//Hour pulses
scConnector.scTwilightData.axHours[0]		:= scConnector.scTwilightData.todSystem = TOD#00:00:00 AND scConnector.scTwilightData.dtSystem <> DT#1970-1-1-00:00:00;	//Fix for startup
scConnector.scTwilightData.axHours[1]		:= scConnector.scTwilightData.todSystem = TOD#01:00:00;
scConnector.scTwilightData.axHours[2]		:= scConnector.scTwilightData.todSystem = TOD#02:00:00;
scConnector.scTwilightData.axHours[3]		:= scConnector.scTwilightData.todSystem = TOD#03:00:00;
scConnector.scTwilightData.axHours[4]		:= scConnector.scTwilightData.todSystem = TOD#04:00:00;
scConnector.scTwilightData.axHours[5]		:= scConnector.scTwilightData.todSystem = TOD#05:00:00;
scConnector.scTwilightData.axHours[6]		:= scConnector.scTwilightData.todSystem = TOD#06:00:00;
scConnector.scTwilightData.axHours[7]		:= scConnector.scTwilightData.todSystem = TOD#07:00:00;
scConnector.scTwilightData.axHours[8]		:= scConnector.scTwilightData.todSystem = TOD#08:00:00;
scConnector.scTwilightData.axHours[9]		:= scConnector.scTwilightData.todSystem = TOD#09:00:00;
scConnector.scTwilightData.axHours[10]		:= scConnector.scTwilightData.todSystem = TOD#10:00:00;
scConnector.scTwilightData.axHours[11]		:= scConnector.scTwilightData.todSystem = TOD#11:00:00;
scConnector.scTwilightData.axHours[12]		:= scConnector.scTwilightData.todSystem = TOD#12:00:00;
scConnector.scTwilightData.axHours[13]		:= scConnector.scTwilightData.todSystem = TOD#13:00:00;
scConnector.scTwilightData.axHours[14]		:= scConnector.scTwilightData.todSystem = TOD#14:00:00;
scConnector.scTwilightData.axHours[15]		:= scConnector.scTwilightData.todSystem = TOD#15:00:00;
scConnector.scTwilightData.axHours[16]		:= scConnector.scTwilightData.todSystem = TOD#16:00:00;
scConnector.scTwilightData.axHours[17]		:= scConnector.scTwilightData.todSystem = TOD#17:00:00;
scConnector.scTwilightData.axHours[18]		:= scConnector.scTwilightData.todSystem = TOD#18:00:00;
scConnector.scTwilightData.axHours[19]		:= scConnector.scTwilightData.todSystem = TOD#19:00:00;
scConnector.scTwilightData.axHours[20]		:= scConnector.scTwilightData.todSystem = TOD#20:00:00;
scConnector.scTwilightData.axHours[21]		:= scConnector.scTwilightData.todSystem = TOD#21:00:00;
scConnector.scTwilightData.axHours[22]		:= scConnector.scTwilightData.todSystem = TOD#22:00:00;
scConnector.scTwilightData.axHours[23]		:= scConnector.scTwilightData.todSystem = TOD#23:00:00;
END_ACTION

{attribute 'monitoring' := 'call'} PROPERTY tSlaveErrorResetTime :TIME
SET
tSlaveErrorResetTime_int := tSlaveErrorResetTime;
END_SET
GET
tSlaveErrorResetTime := tSlaveErrorResetTime_int;
END_GET
END_PROPERTY

METHOD Configure_AutoSyncClock
VAR_INPUT
	xAutoSyncClocks		:BOOL := TRUE;		//Sync system time with server
	tAutoSyncClocks		:TIME := T#3H;		//Time for each sync
END_VAR
xAutoSyncClocks_int := xAutoSyncClocks;
tAutoSyncClocks_int := tAutoSyncClocks;
END_METHOD


METHOD Configure_MQTT
VAR_INPUT
	sMQTT_IPAddress				:STRING(15) := '192.168.1.10';
	uiMQTT_ServerPort			:UINT := 1883;
	sMQTT_Username				:STRING(32);
	sMQTT_Password				:STRING(32);
	tMQTT_UpdateTimeOut			:TIME := T#60S;
END_VAR
sMQTT_IPAddress_int := sMQTT_IPAddress;
uiMQTT_ServerPort_int := uiMQTT_ServerPort;
sMQTT_Username_int := sMQTT_Username;
sMQTT_Password_int := sMQTT_Password;
tMQTT_UpdateTimeOut_int := tMQTT_UpdateTimeOut;
END_METHOD

METHOD Configure_HTTP
VAR_INPUT
	sHTTP_IPAddress			:STRING(15) := '192.168.1.10';
	uiHTTP_ServerPort		:UINT := 8080;
END_VAR
sHTTP_IPAddress_int := sHTTP_IPAddress;
uiHTTP_ServerPort_int := uiHTTP_ServerPort;
END_METHOD

METHOD Configure_Twilight
VAR_INPUT
	todSunOffset		:TOD := TOD#00:30:00;	//Time offset (Pre-sunset) / (Post-sunrise)
	todSystemTime_Offset:TOD := TOD#00:00:00;	//Time offset from server to show correct time on system
END_VAR
todSunOffset_int := todSunOffset;
todSystemTime_Offset_int := todSystemTime_Offset;
END_METHOD

{attribute 'monitoring' := 'call'} PROPERTY xAutoReconnect :BOOL
SET
xAutoReconnect_int := xAutoReconnect;
END_SET
GET
xAutoReconnect := xAutoReconnect_int;
END_GET
END_PROPERTY

{attribute 'monitoring' := 'call'} PROPERTY tDataForceSetValues :TIME
SET
tDataForceSetValues_int := tDataForceSetValues;
END_SET
GET
tDataForceSetValues := tDataForceSetValues_int;
END_GET
END_PROPERTY

{attribute 'monitoring' := 'call'} PROPERTY udiUpdateRate_MQTT :UDINT
GET
udiUpdateRate_MQTT := udiUpdateRate_MQTT_int;
END_GET
END_PROPERTY

{attribute 'monitoring' := 'call'} PROPERTY xStartUpDone :BOOL
GET
xStartUpDone := xHTTP_StartUpDone;
END_GET
END_PROPERTY

ACTION ErrorHandling:
//Write error to output
//Sorted on importance	
{warning disable C0327}
//HTTP (1000+)
IF NOT TON_SlaveError_Reset.IN
AND fbHTTP.xError THEN
	scError.xError := TRUE;
	scError.eErrorID := fbHTTP.eErrorID;
	scError.sErrorInstance := _Domoticz_StringExtractAfterDot(sInstanceName);
	sErrorInstance_Concat := '.fbHTTP';
	scError.sErrorInfo := '';
	
//HTTP JSON (3000+)
//Parsing error
ELSIF NOT TON_SlaveError_Reset.IN
AND fbHTTP_Parser.xError THEN
	scError.xError := TRUE;
	scError.eErrorID := fbHTTP_Parser.eErrorID;
	scError.sErrorInstance := _Domoticz_StringExtractAfterDot(sInstanceName);
	sErrorInstance_Concat := '.fbHTTP_Parser';
	scError.sErrorInfo := '';

//HTTP Update timeout
ELSIF NOT TON_SlaveError_Reset.IN
AND TON_HTTP_UpdateTimeOut.Q THEN
	scError.xError := TRUE;
	scError.eErrorID := Domoticz_eErrors.HTTPUpdateTimeOut;
	scError.sErrorInstance := _Domoticz_StringExtractAfterDot(sInstanceName);
	sErrorInstance_Concat := '';
	scError.sErrorInfo := '';
	
//HTTP Connection lost
ELSIF NOT TON_SlaveError_Reset.IN
AND iStepper_HTTP = -10 THEN
	scError.xError := TRUE;
	scError.eErrorID := Domoticz_eErrors.HTTPConnectionLost;
	scError.sErrorInstance := _Domoticz_StringExtractAfterDot(sInstanceName);
	sErrorInstance_Concat := '';
	scError.sErrorInfo := '';
	
//MQTT Receive (2000+)
ELSIF NOT TON_SlaveError_Reset.IN
AND fbMQTT_Receive.xError THEN
	scError.xError := TRUE;
	scError.eErrorID := fbMQTT_Receive.eErrorID;
	scError.sErrorInstance := _Domoticz_StringExtractAfterDot(sInstanceName);
	sErrorInstance_Concat := '.fbMQTT_Receive';
	scError.sErrorInfo := '';
	
//MQTT Send (2000+)
ELSIF NOT TON_SlaveError_Reset.IN
AND fbMQTT_Send.xError THEN
	scError.xError := TRUE;
	scError.eErrorID := fbMQTT_Send.eErrorID;
	scError.sErrorInstance := _Domoticz_StringExtractAfterDot(sInstanceName);
	sErrorInstance_Concat := '.fbMQTT_Send';
	scError.sErrorInfo := '';
	
//MQTT JSON (3000+)
//Error in parsing
ELSIF NOT TON_SlaveError_Reset.IN
AND fbMQTT_Parser.xError THEN
	scError.xError := TRUE;
	scError.eErrorID := fbMQTT_Parser.eErrorID;
	scError.sErrorInstance := _Domoticz_StringExtractAfterDot(sInstanceName);
	sErrorInstance_Concat := '.fbMQTT_Parser';
	scError.sErrorInfo := '';
	
//MQTT Update timeout
ELSIF NOT TON_SlaveError_Reset.IN
AND TON_MQTT_UpdateTimeOut.Q THEN 
	scError.xError := TRUE;
	scError.eErrorID := Domoticz_eErrors.MQTTUpdateTimeOut;
	scError.sErrorInstance := _Domoticz_StringExtractAfterDot(sInstanceName);
	sErrorInstance_Concat := '';
	scError.sErrorInfo := '';
//MQTT Connection lost
ELSIF NOT TON_SlaveError_Reset.IN
AND iStepper_MQTT = -10 THEN 
	scError.xError := TRUE;
	scError.eErrorID := Domoticz_eErrors.MQTTConnectionLost;
	scError.sErrorInstance := _Domoticz_StringExtractAfterDot(sInstanceName);
	sErrorInstance_Concat := '';
	scError.sErrorInfo := '';
{warning restore C0327}

//Error reading data from HTTP object value
ELSIF NOT TON_SlaveError_Reset.IN
AND xHTTP_ObjectError
AND uiHTTP_ObjectError_Source <> 0
AND uiHTTP_ObjectError_wX <> 0 THEN
	scError.xError := TRUE;
	scError.eErrorID := eHTTP_ObjectError;
	scError.sErrorInstance := _Domoticz_StringExtractAfterDot(sInstanceName);
	sErrorInstance_Concat := '';
	sErrorInstance_Concat := CONCAT('.afbHTTP_Object.uiIdentifier[', 	TO_STRING(uiHTTP_ObjectError_Source));
	sErrorInstance_Concat := CONCAT(sErrorInstance_Concat, 				'].uiIdentifier:');
	sErrorInstance_Concat := CONCAT(sErrorInstance_Concat,				TO_STRING(uiHTTP_ObjectError_wX));
	scError.sErrorInfo := '';
	
//Max amount of slaves connected
ELSIF NOT TON_SlaveError_Reset.IN
AND scConnector.uiSlaveTotal = Domoticz_Properties.uiMaxConnectedSlaves THEN
	scError.xError := TRUE;
	scError.eErrorID := Domoticz_eErrors.ObjectMaxReached;
	scError.sErrorInstance := _Domoticz_StringExtractAfterDot(sInstanceName);
	sErrorInstance_Concat := '';
	scError.sErrorInfo := '';
	
//Post server status when booting
ELSIF NOT xHTTP_StartUpDone THEN
	scError.xError := TRUE;
	scError.eErrorID := Domoticz_eErrors.ServerStarting;
	scError.sErrorInstance := _Domoticz_StringExtractAfterDot(sInstanceName);
	sErrorInstance_Concat := '';
	scError.sErrorInfo := '';
	
	//Also write internal state
	scConnector.scSlaveError.xError	:= TRUE;
	scConnector.scSlaveError.eErrorID := Domoticz_eErrors.ServerStarting;
	scConnector.scSlaveError.sErrorInstance := '';
	scConnector.scSlaveError.sErrorInfo := '';
	
//Delete server startup message
ELSIF xHTTP_StartUpDone 
AND scConnector.scSlaveError.xError
AND scConnector.scSlaveError.eErrorID = Domoticz_eErrors.ServerStarting THEN
	scError := scError_Empty;
	scConnector.scSlaveError := scError_Empty;

//(New) error from slave (only when HTTP update is done once and not yet triggered)
ELSIF xHTTP_StartUpDone 
AND scConnector.scSlaveError.xError
AND scConnector.scSlaveError.eErrorID <> Domoticz_eErrors.NoError
AND scConnector.scSlaveError.udiUniqueID = 0
AND NOT TON_SlaveError_Reset.IN THEN
	//Set timer
	TON_SlaveError_Reset.IN := TRUE;
	//Register, check voor empty space
	FOR wX := 1 TO Domoticz_Properties.uiActiveErrors DO
		IF ascActiveSlaveErrors_int[wX].udiUniqueID = 0 THEN
			ascActiveSlaveErrors_int[wX] := scConnector.scSlaveError;
			{warning disable C0371}
			ascActiveSlaveErrors_int[wX].udiUniqueID := TO_UDINT(scConnector.scTwilightData.dtSystem);
			{warning restore C0371}
			scConnector.scSlaveError.udiUniqueID := ascActiveSlaveErrors_int[wX].udiUniqueID;
			EXIT;
		END_IF
	END_FOR
	//End of array reached, no place available
	IF wX = (Domoticz_Properties.uiActiveErrors+1) THEN
		//Return result invalid
		scError.xError := TRUE;
		scError.eErrorID := Domoticz_eErrors.ErrorHandlerArrayFull;
		scError.sErrorInstance := _Domoticz_StringExtractAfterDot(sInstanceName);
		scError.sErrorInfo := '';
		sErrorInstance_Concat := '';
		//scConnector.scSlaveError.udiUniqueID := 0;	//Delete response > no feedback to ErrorInterface FB
	END_IF
	//Output
	scError := scConnector.scSlaveError;	//Copy
	sErrorInstance_Concat := '';	//No additional info
	
//(Remove) error from slave
ELSIF xHTTP_StartUpDone
AND scConnector.scSlaveError.xError
AND scConnector.scSlaveError.eErrorID = Domoticz_eErrors.NoError
AND scConnector.scSlaveError.udiUniqueID <> 0 THEN
	//Unregister, look for ID
	FOR wX := 1 TO Domoticz_Properties.uiActiveErrors DO
		IF ascActiveSlaveErrors_int[wX].udiUniqueID = scConnector.scSlaveError.udiUniqueID THEN
			//Delete entry anyhow
			ascActiveSlaveErrors_int[wX] := scError_Empty;
			//Shift upper array elements
			IF wX <= (Domoticz_Properties.uiActiveErrors-1) THEN
				FOR wY := wX TO (Domoticz_Properties.uiActiveErrors-1) DO
					ascActiveSlaveErrors_int[wY] := ascActiveSlaveErrors_int[wY+1];
				END_FOR
			END_IF
			//Clean last element
			ascActiveSlaveErrors_int[Domoticz_Properties.uiActiveErrors] := scError_Empty;
			EXIT;
		END_IF
	END_FOR
	//End of array reached, not found
	IF wX = (Domoticz_Properties.uiActiveErrors+1) THEN
		//Return result invalid
		scError.xError := TRUE;
		scError.eErrorID := Domoticz_eErrors.ErrorHandlerEntryNotFound;
		scError.sErrorInstance := _Domoticz_StringExtractAfterDot(sInstanceName);
		scError.sErrorInfo := '';
		sErrorInstance_Concat := '';
	END_IF
	//Clear output and connector
	scError := scError_Empty;
	scConnector.scSlaveError := scError_Empty;

//Remove slave error from output after set time
ELSIF xHTTP_StartUpDone 
AND TON_SlaveError_Reset.IN
AND TON_SlaveError_Reset.Q THEN
	//Reset timer
	TON_SlaveError_Reset.IN := FALSE;
	//Clear output and connector
	scError := scError_Empty;
	scConnector.scSlaveError := scError_Empty;
	
//No errors
ELSIF NOT TON_SlaveError_Reset.IN THEN
	scError.xError := FALSE;
	scError.eErrorID := Domoticz_eErrors.NoError;
	scError.sErrorInstance := '';
	sErrorInstance_Concat := '';
	scError.sErrorInfo := '';
END_IF

TON_SlaveError_Reset(IN:=, PT:=tSlaveErrorResetTime_int);	//Run reset timer

//Concat extra source information if available, delete afterwards
psErrorInstance := ADR(scError.sErrorInstance);
psErrorInstance_Concat := ADR(sErrorInstance_Concat);
IF sErrorInstance_Concat <> '' THEN
	StrConcatA(psErrorInstance_Concat, psErrorInstance, SIZEOF(scError.sErrorInstance));
	sErrorInstance_Concat := '';
END_IF
END_ACTION

PROPERTY ascActiveSlaveErrors :ARRAY[1..Domoticz_Properties.uiActiveErrors] OF Domoticz_scError;
GET
ascActiveSlaveErrors := ascActiveSlaveErrors_int;
END_GET
END_PROPERTY

END_FUNCTION_BLOCK

// Function Blocks/Server/_Domoticz_Server_HTTP_Object
{attribute 'conditionalshow_all_locals'}
{attribute 'conditionalshow'}
FUNCTION_BLOCK _Domoticz_Server_HTTP_Object
VAR_INPUT
	sIPAddress					:STRING(15) := '192.168.1.10';
	uiServerPort				:UINT := 8080;
	tTimeOut					:TIME := T#3S;
	dtTimeStamp					:DT;
	xReadData					:BOOL;
	uiIdentifier				:UINT;
END_VAR
VAR_OUTPUT
	xError						:BOOL;
	eErrorID					:Domoticz_eErrors;
	xBusy						:BOOL;
	xDone						:BOOL;
	scObjectData				:Domoticz_scObjectData;
END_VAR
VAR
	//Internal          	
	wX							:WORD;
	xReadData_mem				:BOOL;
	       	
	iStepper					:INT;
	fbHTTP						:SNDLTN_HTTP.HTTP_Client;
	xHTTP_TypeMatched			:BOOL;
	                        	
	xHTTP_DataError				:BOOL;		//Received data contains error
	iHTTP_DataError				:INT;		//Count data errors
	
	//Used for concatting values
	sHTTP_Concat				:STRING(SNDLTN_HTTP.HTTP_Properties.uiHTTPMaxURLSize);
	psHTTP_Concat				:POINTER TO STRING(SNDLTN_HTTP.HTTP_Properties.uiHTTPMaxURLSize);
	sHTTP_ConcatHelper			:STRING(SNDLTN_HTTP.HTTP_Properties.uiHTTPMaxURLSize);
	psHTTP_ConcatHelper			:POINTER TO STRING(SNDLTN_HTTP.HTTP_Properties.uiHTTPMaxURLSize);
	                        	
	//JSON	                	
	fbHTTP_Parser				:SNDLTN_JSON.JSON_Parser;
	fbHTTP_Values				:SNDLTN_JSON.JSON_GetMultiValue;
	
	eHTTP_HumidityStatus		:Domoticz_eHumidityStatus;

END_VAR

Main();

ACTION Main:
{attribute 'conditionalshow'}
CASE iStepper OF

	-10:	//Error
			
		//Reset if needed
		IF NOT xReadData_mem THEN
			xError := FALSE;
			fbHTTP_Parser.xResetError := TRUE;
			iStepper := 0;
		END_IF
	
	0:	//Disabled
		
		//Set outputs if not used
		IF NOT xReadData_mem THEN
			ResetObjectData(); //Empty output
			xBusy := FALSE;
			xDone := FALSE;
		END_IF
		
		//Reset commands
		fbHTTP.xExecute := FALSE;
		fbHTTP_Parser.xResetError := FALSE;
		iHTTP_DataError := 0;
		
		//Wait for command
		IF xReadData AND NOT xReadData_mem
		AND uiIdentifier <> 0 THEN
			xBusy := TRUE;
			iStepper := 10;
		//Invalid identifier
		ELSIF xReadData AND NOT xReadData_mem
		AND uiIdentifier = 0 THEN
			xError := TRUE;
			eErrorID := Domoticz_eErrors.HTTP_InvalidIdentifier;
			iStepper := -10;
		END_IF
		
	10:	//Update object
		
		//Execute and process data
		fbHTTP.xExecute := TRUE;
		DataObject_In();	//Process data
		
		//Wait until processed
		//Not all data received, retrigger
		IF (fbHTTP.xDone AND NOT fbHTTP.xResponseValid) OR xHTTP_DataError THEN
			xHTTP_DataError := FALSE;
			fbHTTP.xExecute := FALSE;
			iHTTP_DataError := iHTTP_DataError + 1;
		//Retrigger max reached, continue (probably invalid ID?)
		ELSIF iHTTP_DataError > 5 THEN
			fbHTTP.xExecute := FALSE;
			xBusy := FALSE;
			xDone := FALSE;
			iStepper := -10;		
		//All data received, continue
		ELSIF fbHTTP.xDone AND fbHTTP.xResponseValid THEN
			fbHTTP.xExecute := FALSE;
			xBusy := FALSE;
			xDone := TRUE;
			iStepper := 0;
		END_IF
		
		//Error occured (outputted in main)
		IF fbHTTP.xError THEN
			xError := TRUE;
			{warning disable C0327}
			eErrorID := fbHTTP.eErrorID;
			{warning restore C0327}
			iStepper := -10;
		ELSIF fbHTTP_Parser.xError THEN
			xError := TRUE;
			eErrorID := Domoticz_eErrors.HTTP_ParsingError;
			iStepper := -10;
		END_IF
	
END_CASE


//HTTP Server
fbHTTP(
	xExecute:= , 
	udiTimeOut:= TIME_TO_UDINT(tTimeOut)*1000, 
);

//Parse HTTP content > only processed if input changes
fbHTTP_Parser(
	xResetError:= , 
	sContent:= fbHTTP.scResponse.sContent, 
);
	
//Get JSON values
fbHTTP_Values(
	pasProperties:= ADR(fbHTTP_Parser.asProperties[0,0]), 
	asPropertyName:= , 
	aeConversionType:= , 
);

//Mem input
xReadData_mem := xReadData;
END_ACTION

METHOD ResetObjectData
VAR_INPUT
END_VAR
scObjectData.uiIdentifier		:= 0;
scObjectData.dtLastUpdate		:= DT#1970-1-1-00:00:00;
scObjectData.dtTimeStamp		:= DT#1970-1-1-00:00:00;
FOR wX := 1 TO Domoticz_Constants.uiMaxSValues DO
	scObjectData.asValue[wX]	:= '';
END_FOR
scObjectData.iValue				:= 0;
scObjectData.eSource			:= _Domoticz_eDataSource.All;
scObjectData.eCommand			:=_Domoticz_eCommandType.Default;
scObjectData.sDeviceType		:= '';
END_METHOD

ACTION DataObject_In:
{attribute 'conditionalshow'}
//HTTP

//Get pointers
psHTTP_Concat := ADR(sHTTP_Concat);
psHTTP_ConcatHelper := ADR(sHTTP_ConcatHelper);

//Construct URL

//HTTP://
sHTTP_Concat := Domoticz_Constants.sURL_HTTP;

//Add server IP
StrConcatA(ADR(sIPAddress), psHTTP_Concat, TO_INT(SNDLTN_HTTP.HTTP_Properties.uiHTTPMaxURLSize));

//Add seperator
sHTTP_ConcatHelper := ':';
StrConcatA(psHTTP_ConcatHelper, psHTTP_Concat, TO_INT(SNDLTN_HTTP.HTTP_Properties.uiHTTPMaxURLSize));

//Add server port
sHTTP_ConcatHelper := TO_STRING(uiServerPort);
StrConcatA(psHTTP_ConcatHelper, psHTTP_Concat, TO_INT(SNDLTN_HTTP.HTTP_Properties.uiHTTPMaxURLSize));

//Add request
StrConcatA(ADR(Domoticz_Constants.sURL_Object), psHTTP_Concat, TO_INT(SNDLTN_HTTP.HTTP_Properties.uiHTTPMaxURLSize));

//Add identifier
sHTTP_ConcatHelper := TO_STRING(uiIdentifier);
StrConcatA(psHTTP_ConcatHelper, psHTTP_Concat, TO_INT(SNDLTN_HTTP.HTTP_Properties.uiHTTPMaxURLSize));

//Get data from HTTP/JSON
fbHTTP.sURL := sHTTP_Concat;
fbHTTP.eRequestType := HTTP_eRequestType.GET;

//Specify data

//Type
fbHTTP_Values.asPropertyName[_Domoticz_eHTTP_PropertyNames.ObjectType] 			:= Domoticz_Constants.sPropertyHTTP_Type;
fbHTTP_Values.aeConversionType[_Domoticz_eHTTP_PropertyNames.ObjectType] 			:= JSON_eConversionType.None;
//Data                                  						                    
fbHTTP_Values.asPropertyName[_Domoticz_eHTTP_PropertyNames.Data] 					:= Domoticz_Constants.sPropertyHTTP_Data;
fbHTTP_Values.aeConversionType[_Domoticz_eHTTP_PropertyNames.Data] 				:= JSON_eConversionType.None;
//SwitchType                            						                    
fbHTTP_Values.asPropertyName[_Domoticz_eHTTP_PropertyNames.SwitchType] 			:= Domoticz_Constants.sPropertyHTTP_SwitchType;
fbHTTP_Values.aeConversionType[_Domoticz_eHTTP_PropertyNames.SwitchType] 			:= JSON_eConversionType.None;
//LastUpdate                            						                    
fbHTTP_Values.asPropertyName[_Domoticz_eHTTP_PropertyNames.LastUpdate] 			:= Domoticz_Constants.sPropertyHTTP_LastUpdate;
fbHTTP_Values.aeConversionType[_Domoticz_eHTTP_PropertyNames.LastUpdate] 			:= JSON_eConversionType.DateAndTime;
                                        						                    
//Level                                 						                    
fbHTTP_Values.asPropertyName[_Domoticz_eHTTP_PropertyNames.Level] 					:= Domoticz_Constants.sPropertyHTTP_Level;
fbHTTP_Values.aeConversionType[_Domoticz_eHTTP_PropertyNames.Level] 				:= JSON_eConversionType.None;
                                        						                                                          						                    
//Additional                            						                    
//Temp+hum+baro                         						                    
//Temperature                           						                    
fbHTTP_Values.asPropertyName[_Domoticz_eHTTP_PropertyNames.Temperature] 			:= Domoticz_Constants.sPropertyHTTP_Temperature;
fbHTTP_Values.aeConversionType[_Domoticz_eHTTP_PropertyNames.Temperature] 			:= JSON_eConversionType.None;
//Humidity                              						                    
fbHTTP_Values.asPropertyName[_Domoticz_eHTTP_PropertyNames.Humidity] 				:= Domoticz_Constants.sPropertyHTTP_Humidity;
fbHTTP_Values.aeConversionType[_Domoticz_eHTTP_PropertyNames.Humidity] 			:= JSON_eConversionType.None;
//Humidity status                           						                    
fbHTTP_Values.asPropertyName[_Domoticz_eHTTP_PropertyNames.HumidityStatus] 		:= Domoticz_Constants.sPropertyHTTP_HumidityStatus;
fbHTTP_Values.aeConversionType[_Domoticz_eHTTP_PropertyNames.HumidityStatus] 		:= JSON_eConversionType.None;
//Barometer                             						                    
fbHTTP_Values.asPropertyName[_Domoticz_eHTTP_PropertyNames.Barometer] 				:= Domoticz_Constants.sPropertyHTTP_Barometer;
fbHTTP_Values.aeConversionType[_Domoticz_eHTTP_PropertyNames.Barometer] 			:= JSON_eConversionType.None;
//Forecast                    						                    
fbHTTP_Values.asPropertyName[_Domoticz_eHTTP_PropertyNames.Forecast] 				:= Domoticz_Constants.sPropertyHTTP_Forecast;
fbHTTP_Values.aeConversionType[_Domoticz_eHTTP_PropertyNames.Forecast] 			:= JSON_eConversionType.None;
//DewPoint                              						                    
fbHTTP_Values.asPropertyName[_Domoticz_eHTTP_PropertyNames.DewPoint] 				:= Domoticz_Constants.sPropertyHTTP_DewPoint;
fbHTTP_Values.aeConversionType[_Domoticz_eHTTP_PropertyNames.DewPoint] 			:= JSON_eConversionType.None;
                                        						                    
//Wind                                  						                    
//Speed                                 						                    
fbHTTP_Values.asPropertyName[_Domoticz_eHTTP_PropertyNames.Speed] 					:= Domoticz_Constants.sPropertyHTTP_Speed;
fbHTTP_Values.aeConversionType[_Domoticz_eHTTP_PropertyNames.Speed] 				:= JSON_eConversionType.None;
//Chill                                 						                    
fbHTTP_Values.asPropertyName[_Domoticz_eHTTP_PropertyNames.Chill] 					:= Domoticz_Constants.sPropertyHTTP_Chill;
fbHTTP_Values.aeConversionType[_Domoticz_eHTTP_PropertyNames.Chill] 				:= JSON_eConversionType.None;
//Gust                                  						                    
fbHTTP_Values.asPropertyName[_Domoticz_eHTTP_PropertyNames.Gust] 					:= Domoticz_Constants.sPropertyHTTP_Gust;
fbHTTP_Values.aeConversionType[_Domoticz_eHTTP_PropertyNames.Gust] 				:= JSON_eConversionType.None;
//Direction                             						                    
fbHTTP_Values.asPropertyName[_Domoticz_eHTTP_PropertyNames.Direction] 				:= Domoticz_Constants.sPropertyHTTP_Direction;
fbHTTP_Values.aeConversionType[_Domoticz_eHTTP_PropertyNames.Direction] 			:= JSON_eConversionType.None;
                                        						                    
//Rain                                  						                    
//Rain                                  						                    
fbHTTP_Values.asPropertyName[_Domoticz_eHTTP_PropertyNames.Rain] 					:= Domoticz_Constants.sPropertyHTTP_Rain;
fbHTTP_Values.aeConversionType[_Domoticz_eHTTP_PropertyNames.Rain] 				:= JSON_eConversionType.None;
//RainRate                              						                    
fbHTTP_Values.asPropertyName[_Domoticz_eHTTP_PropertyNames.RainRate] 				:= Domoticz_Constants.sPropertyHTTP_RainRate;
fbHTTP_Values.aeConversionType[_Domoticz_eHTTP_PropertyNames.RainRate] 			:= JSON_eConversionType.None;
                                        						                    
//RGB(W)(W)                             						                    
//Color                                 						                    
fbHTTP_Values.asPropertyName[_Domoticz_eHTTP_PropertyNames.Color] 					:= Domoticz_Constants.sPropertyHTTP_Color;
fbHTTP_Values.aeConversionType[_Domoticz_eHTTP_PropertyNames.Color] 				:= JSON_eConversionType.None;
                                        						                    
//Energy                                						                    
//Counter cumulative                    						                    
fbHTTP_Values.asPropertyName[_Domoticz_eHTTP_PropertyNames.Counter] 				:= Domoticz_Constants.sPropertyHTTP_Counter;
fbHTTP_Values.aeConversionType[_Domoticz_eHTTP_PropertyNames.Counter] 				:= JSON_eConversionType.None;
//Counter today                     					                        
fbHTTP_Values.asPropertyName[_Domoticz_eHTTP_PropertyNames.CounterToday] 			:= Domoticz_Constants.sPropertyHTTP_CounterToday;
fbHTTP_Values.aeConversionType[_Domoticz_eHTTP_PropertyNames.CounterToday]			:= JSON_eConversionType.None;
//Counter delivery cumulative           						                    
fbHTTP_Values.asPropertyName[_Domoticz_eHTTP_PropertyNames.CounterDelivery] 		:= Domoticz_Constants.sPropertyHTTP_CounterDelivery;
fbHTTP_Values.aeConversionType[_Domoticz_eHTTP_PropertyNames.CounterDelivery] 		:= JSON_eConversionType.None;
//Counter delivery today                  					                        
fbHTTP_Values.asPropertyName[_Domoticz_eHTTP_PropertyNames.CounterDeliveryToday] 	:= Domoticz_Constants.sPropertyHTTP_CounterDeliveryToday;
fbHTTP_Values.aeConversionType[_Domoticz_eHTTP_PropertyNames.CounterDeliveryToday]	:= JSON_eConversionType.None;
//Usage                                 						                    
fbHTTP_Values.asPropertyName[_Domoticz_eHTTP_PropertyNames.Usage] 					:= Domoticz_Constants.sPropertyHTTP_Usage;
fbHTTP_Values.aeConversionType[_Domoticz_eHTTP_PropertyNames.Usage] 				:= JSON_eConversionType.None;
//Usage delivery                        					                        
fbHTTP_Values.asPropertyName[_Domoticz_eHTTP_PropertyNames.UsageDelivery] 			:= Domoticz_Constants.sPropertyHTTP_UsageDelivery;
fbHTTP_Values.aeConversionType[_Domoticz_eHTTP_PropertyNames.UsageDelivery]		:= JSON_eConversionType.None;

//Reset data on start
IF NOT fbHTTP.xDone THEN
	FOR wX := 1 TO Domoticz_Constants.uiMaxSValues DO
		scObjectData.asValue[wX] := '';
	END_FOR		
END_IF
//******************************************************************JSON:PARSE
IF fbHTTP.xDone AND fbHTTP.xResponseValid THEN
		
	scObjectData.uiIdentifier := uiIdentifier;
	
	//Reset data
	FOR wX := 1 TO Domoticz_Constants.uiMaxSValues DO
		scObjectData.asValue[wX] := '';
	END_FOR
	scObjectData.iValue := 0;
	xHTTP_TypeMatched := FALSE;
	
	//Select correct types
	//Switch
	IF fbHTTP_Values.axMatchFound[_Domoticz_eHTTP_PropertyNames.ObjectType] 
	AND (fbHTTP_Values.asPropertyValue[_Domoticz_eHTTP_PropertyNames.ObjectType] = Domoticz_Constants.sType_Lighting1
	OR fbHTTP_Values.asPropertyValue[_Domoticz_eHTTP_PropertyNames.ObjectType] = Domoticz_Constants.sType_Lighting2
	OR fbHTTP_Values.asPropertyValue[_Domoticz_eHTTP_PropertyNames.ObjectType] = Domoticz_Constants.sType_Lighting3
	OR fbHTTP_Values.asPropertyValue[_Domoticz_eHTTP_PropertyNames.ObjectType] = Domoticz_Constants.sType_Lighting4
	OR fbHTTP_Values.asPropertyValue[_Domoticz_eHTTP_PropertyNames.ObjectType] = Domoticz_Constants.sType_Lighting5
	OR fbHTTP_Values.asPropertyValue[_Domoticz_eHTTP_PropertyNames.ObjectType] = Domoticz_Constants.sType_LightSwitch
	OR fbHTTP_Values.asPropertyValue[_Domoticz_eHTTP_PropertyNames.ObjectType] = Domoticz_Constants.sType_Security) THEN
		xHTTP_TypeMatched := TRUE;
		//Selector or selector switch
		IF fbHTTP_Values.axMatchFound[_Domoticz_eHTTP_PropertyNames.SwitchType] 
		AND (fbHTTP_Values.asPropertyValue[_Domoticz_eHTTP_PropertyNames.SwitchType] = Domoticz_Constants.sSwitchType_Selector
		OR fbHTTP_Values.asPropertyValue[_Domoticz_eHTTP_PropertyNames.SwitchType] = Domoticz_Constants.sSwitchType_SelectorSwitch) THEN	
			IF fbHTTP_Values.axMatchFound[_Domoticz_eHTTP_PropertyNames.Level] THEN	//Level
				scObjectData.iValue := 2; 
				scObjectData.asValue[Domoticz_eSValues_General.General] := TO_STRING(_Domoticz_StringToReal(fbHTTP_Values.asPropertyValue[_Domoticz_eHTTP_PropertyNames.Level])); 	//Remove any values				
			ELSIF fbHTTP_Values.axMatchFound[_Domoticz_eHTTP_PropertyNames.Data] THEN	//Data
				scObjectData.iValue := 2; 
				scObjectData.asValue[Domoticz_eSValues_General.General] := TO_STRING(_Domoticz_StringToReal(fbHTTP_Values.asPropertyValue[_Domoticz_eHTTP_PropertyNames.Data])); 	//Remove any values
			END_IF
		//Dimmer
		ELSIF fbHTTP_Values.axMatchFound[_Domoticz_eHTTP_PropertyNames.SwitchType] 
		AND fbHTTP_Values.asPropertyValue[_Domoticz_eHTTP_PropertyNames.SwitchType] = Domoticz_Constants.sSwitchType_Dimmer THEN
			IF fbHTTP_Values.axMatchFound[_Domoticz_eHTTP_PropertyNames.Level] THEN	//Data / Set level
				IF fbHTTP_Values.axMatchFound[_Domoticz_eHTTP_PropertyNames.Data] 
				AND TO_BOOL(_Domoticz_StringToByte(fbHTTP_Values.asPropertyValue[_Domoticz_eHTTP_PropertyNames.Data])) THEN//Dimmer turned off
					scObjectData.iValue := 2; 
					scObjectData.asValue[Domoticz_eSValues_General.General] := TO_STRING(_Domoticz_StringToReal(fbHTTP_Values.asPropertyValue[_Domoticz_eHTTP_PropertyNames.Level])); 	//Remove any values
				ELSE
					IF fbHTTP_Values.axMatchFound[_Domoticz_eHTTP_PropertyNames.Data] THEN		//Data
						scObjectData.iValue := TO_INT(_Domoticz_StringToByte(fbHTTP_Values.asPropertyValue[_Domoticz_eHTTP_PropertyNames.Data])); 
					END_IF
				END_IF
			END_IF
		//None of above
		ELSE	
			IF fbHTTP_Values.axMatchFound[_Domoticz_eHTTP_PropertyNames.Data] THEN 	//Data
				scObjectData.iValue := TO_INT(_Domoticz_StringToByte(fbHTTP_Values.asPropertyValue[_Domoticz_eHTTP_PropertyNames.Data])); 
			END_IF
		END_IF
		
	//RGB(W)(W)
	ELSIF fbHTTP_Values.axMatchFound[_Domoticz_eHTTP_PropertyNames.ObjectType] 
	AND fbHTTP_Values.asPropertyValue[_Domoticz_eHTTP_PropertyNames.ObjectType] = Domoticz_Constants.sType_ColorSwitch THEN
		xHTTP_TypeMatched := TRUE;
		//Color settings
		IF fbHTTP_Values.axMatchFound[_Domoticz_eHTTP_PropertyNames.Color] THEN //Color
			scObjectData.asValue[Domoticz_eSValues_Colors.Red] 			:= _Domoticz_StringExtractColor(fbHTTP_Values.asPropertyValue[_Domoticz_eHTTP_PropertyNames.Color], Domoticz_eSValues_Colors.Red); 
			scObjectData.asValue[Domoticz_eSValues_Colors.Green] 		:= _Domoticz_StringExtractColor(fbHTTP_Values.asPropertyValue[_Domoticz_eHTTP_PropertyNames.Color], Domoticz_eSValues_Colors.Green);
			scObjectData.asValue[Domoticz_eSValues_Colors.Blue] 		:= _Domoticz_StringExtractColor(fbHTTP_Values.asPropertyValue[_Domoticz_eHTTP_PropertyNames.Color], Domoticz_eSValues_Colors.Blue);
			scObjectData.asValue[Domoticz_eSValues_Colors.ColdWhite]	:= _Domoticz_StringExtractColor(fbHTTP_Values.asPropertyValue[_Domoticz_eHTTP_PropertyNames.Color], Domoticz_eSValues_Colors.ColdWhite);
			scObjectData.asValue[Domoticz_eSValues_Colors.WarmWhite]	:= _Domoticz_StringExtractColor(fbHTTP_Values.asPropertyValue[_Domoticz_eHTTP_PropertyNames.Color], Domoticz_eSValues_Colors.WarmWhite);
		END_IF	
		//Brightness level
		IF fbHTTP_Values.axMatchFound[_Domoticz_eHTTP_PropertyNames.Level] THEN //Level (from 0-100 to 0-255)
			scObjectData.asValue[Domoticz_eSValues_Colors.Brightness] := TO_STRING(TRUNC(_Domoticz_StringToReal(fbHTTP_Values.asPropertyValue[_Domoticz_eHTTP_PropertyNames.Level])));
		END_IF
		//Check 'OFF' status
		IF fbHTTP_Values.axMatchFound[_Domoticz_eHTTP_PropertyNames.Data] THEN 
			scObjectData.iValue := TO_INT(TRUNC(_Domoticz_StringToByte(fbHTTP_Values.asPropertyValue[_Domoticz_eHTTP_PropertyNames.Data])));
			IF scObjectData.iValue = 0 THEN	//Force brightness to zero when not enabled
 				scObjectData.asValue[Domoticz_eSValues_Colors.Brightness] := '0.0';
			END_IF
		END_IF
	
	//Temperature / Humidity / Barometer / Dewpoint
	ELSIF fbHTTP_Values.axMatchFound[_Domoticz_eHTTP_PropertyNames.ObjectType] 
	AND (fbHTTP_Values.asPropertyValue[_Domoticz_eHTTP_PropertyNames.ObjectType] = Domoticz_Constants.sType_Temperature
	OR fbHTTP_Values.asPropertyValue[_Domoticz_eHTTP_PropertyNames.ObjectType] = Domoticz_Constants.sType_TemperatureBaro
	OR fbHTTP_Values.asPropertyValue[_Domoticz_eHTTP_PropertyNames.ObjectType] = Domoticz_Constants.sType_TemperatureHumidity
	OR fbHTTP_Values.asPropertyValue[_Domoticz_eHTTP_PropertyNames.ObjectType] = Domoticz_Constants.sType_TemperatureHumidityBaro
	OR fbHTTP_Values.asPropertyValue[_Domoticz_eHTTP_PropertyNames.ObjectType] = Domoticz_Constants.sType_Humidity) THEN
		xHTTP_TypeMatched := TRUE;
		IF fbHTTP_Values.axMatchFound[_Domoticz_eHTTP_PropertyNames.Temperature] THEN	//Temperature
			scObjectData.asValue[Domoticz_eSValues_TempHumBaro.Temperature] := fbHTTP_Values.asPropertyValue[_Domoticz_eHTTP_PropertyNames.Temperature]; 
		END_IF
		IF fbHTTP_Values.axMatchFound[_Domoticz_eHTTP_PropertyNames.Humidity] THEN		//Humidity
			scObjectData.asValue[Domoticz_eSValues_TempHumBaro.Humidity] := fbHTTP_Values.asPropertyValue[_Domoticz_eHTTP_PropertyNames.Humidity]; 
			scObjectData.iValue := TO_INT(_Domoticz_StringToReal(fbHTTP_Values.asPropertyValue[_Domoticz_eHTTP_PropertyNames.Humidity])); 
		END_IF	
		IF fbHTTP_Values.axMatchFound[_Domoticz_eHTTP_PropertyNames.HumidityStatus] THEN	//Humidity Status
			FOR wX := 0 TO 3 DO
				eHTTP_HumidityStatus := TO_INT(wX);
				IF fbHTTP_Values.asPropertyValue[_Domoticz_eHTTP_PropertyNames.HumidityStatus] = TO_STRING(eHTTP_HumidityStatus) THEN
					scObjectData.asValue[Domoticz_eSValues_TempHumBaro.HumidityStatus] := TO_STRING(TO_INT(eHTTP_HumidityStatus));
					EXIT;
				END_IF
			END_FOR
		END_IF
		IF fbHTTP_Values.axMatchFound[_Domoticz_eHTTP_PropertyNames.Barometer] THEN	//Barometer
			scObjectData.asValue[Domoticz_eSValues_TempHumBaro.Barometer] := fbHTTP_Values.asPropertyValue[_Domoticz_eHTTP_PropertyNames.Barometer]; 
		END_IF
		IF fbHTTP_Values.axMatchFound[_Domoticz_eHTTP_PropertyNames.Barometer] THEN	//Forecast
			scObjectData.asValue[Domoticz_eSValues_TempHumBaro.Forecast] := fbHTTP_Values.asPropertyValue[_Domoticz_eHTTP_PropertyNames.Forecast];
		END_IF 
		IF fbHTTP_Values.axMatchFound[_Domoticz_eHTTP_PropertyNames.DewPoint] THEN		//Dewpoint
			scObjectData.asValue[Domoticz_eSValues_TempHumBaro.DewPoint] := fbHTTP_Values.asPropertyValue[_Domoticz_eHTTP_PropertyNames.DewPoint];
		END_IF
		
	//Air Quality
	ELSIF fbHTTP_Values.axMatchFound[_Domoticz_eHTTP_PropertyNames.ObjectType] 
	AND fbHTTP_Values.asPropertyValue[_Domoticz_eHTTP_PropertyNames.ObjectType] = Domoticz_Constants.sType_AirQuality THEN
		xHTTP_TypeMatched := TRUE;
		IF fbHTTP_Values.axMatchFound[_Domoticz_eHTTP_PropertyNames.Data] THEN		//Data
			scObjectData.iValue := TO_INT(_Domoticz_StringToReal(fbHTTP_Values.asPropertyValue[_Domoticz_eHTTP_PropertyNames.Data])); 
		END_IF
		
	//Wind	
	ELSIF fbHTTP_Values.axMatchFound[_Domoticz_eHTTP_PropertyNames.ObjectType] 
	AND fbHTTP_Values.asPropertyValue[_Domoticz_eHTTP_PropertyNames.ObjectType] = Domoticz_Constants.sType_Wind THEN
		xHTTP_TypeMatched := TRUE;
		IF fbHTTP_Values.axMatchFound[_Domoticz_eHTTP_PropertyNames.Speed] THEN 	//Speed
			scObjectData.asValue[Domoticz_eSValues_Wind.Speed] := fbHTTP_Values.asPropertyValue[_Domoticz_eHTTP_PropertyNames.Speed]; 
		END_IF
		IF fbHTTP_Values.axMatchFound[_Domoticz_eHTTP_PropertyNames.Chill] THEN	//Chill
			scObjectData.asValue[Domoticz_eSValues_Wind.Chill] := fbHTTP_Values.asPropertyValue[_Domoticz_eHTTP_PropertyNames.Chill]; 
		END_IF
		IF fbHTTP_Values.axMatchFound[_Domoticz_eHTTP_PropertyNames.Gust] THEN 	//Gust
			scObjectData.asValue[Domoticz_eSValues_Wind.Gust] := fbHTTP_Values.asPropertyValue[_Domoticz_eHTTP_PropertyNames.Gust]; 
		END_IF
		IF fbHTTP_Values.axMatchFound[_Domoticz_eHTTP_PropertyNames.Direction] THEN	//Direction
			scObjectData.asValue[5] := fbHTTP_Values.asPropertyValue[_Domoticz_eHTTP_PropertyNames.Direction]; 
		END_IF	
		
	//Rain
	ELSIF fbHTTP_Values.axMatchFound[_Domoticz_eHTTP_PropertyNames.ObjectType] 
	AND fbHTTP_Values.asPropertyValue[_Domoticz_eHTTP_PropertyNames.ObjectType] = Domoticz_Constants.sType_Rain THEN
		xHTTP_TypeMatched := TRUE;
		IF fbHTTP_Values.axMatchFound[_Domoticz_eHTTP_PropertyNames.Rain] THEN 	//Rain
			scObjectData.asValue[Domoticz_eSValues_Rain.Rain] := fbHTTP_Values.asPropertyValue[_Domoticz_eHTTP_PropertyNames.Rain]; 
		END_IF
		IF fbHTTP_Values.axMatchFound[_Domoticz_eHTTP_PropertyNames.RainRate] THEN 	//Rain rate
			scObjectData.asValue[Domoticz_eSValues_Rain.RainRate] := fbHTTP_Values.asPropertyValue[_Domoticz_eHTTP_PropertyNames.RainRate]; 
		END_IF	
		
	//P1 Smart Meter
	ELSIF (fbHTTP_Values.axMatchFound[_Domoticz_eHTTP_PropertyNames.ObjectType] 
	AND fbHTTP_Values.asPropertyValue[_Domoticz_eHTTP_PropertyNames.ObjectType] = Domoticz_Constants.sType_P1SmartMeter) THEN
		xHTTP_TypeMatched := TRUE;
		IF fbHTTP_Values.axMatchFound[_Domoticz_eHTTP_PropertyNames.Counter] THEN 	//Power cumulative
			scObjectData.asValue[Domoticz_eSValues_P1.Usage1Cumulative] := fbHTTP_Values.asPropertyValue[_Domoticz_eHTTP_PropertyNames.Counter]; 
		END_IF
		IF fbHTTP_Values.axMatchFound[_Domoticz_eHTTP_PropertyNames.CounterToday] THEN 	//Power today
			scObjectData.asValue[Domoticz_eSValues_P1.UsageToday] := fbHTTP_Values.asPropertyValue[_Domoticz_eHTTP_PropertyNames.CounterToday]; 
		END_IF
		IF fbHTTP_Values.axMatchFound[_Domoticz_eHTTP_PropertyNames.CounterDelivery] THEN 	//Power delivery cumulative
			scObjectData.asValue[Domoticz_eSValues_P1.Return1Cumulative] := fbHTTP_Values.asPropertyValue[_Domoticz_eHTTP_PropertyNames.CounterDelivery]; 
		END_IF
		IF fbHTTP_Values.axMatchFound[_Domoticz_eHTTP_PropertyNames.CounterDeliveryToday] THEN 	//Power delivery today
			scObjectData.asValue[Domoticz_eSValues_P1.ReturnToday] := fbHTTP_Values.asPropertyValue[_Domoticz_eHTTP_PropertyNames.CounterDeliveryToday];
		END_IF 
		IF fbHTTP_Values.axMatchFound[_Domoticz_eHTTP_PropertyNames.Usage] THEN 	//Usage
			scObjectData.asValue[Domoticz_eSValues_P1.UsageActual] := fbHTTP_Values.asPropertyValue[_Domoticz_eHTTP_PropertyNames.Usage]; 
		END_IF
		IF fbHTTP_Values.axMatchFound[_Domoticz_eHTTP_PropertyNames.UsageDelivery] THEN 	//Usage delivery
			scObjectData.asValue[Domoticz_eSValues_P1.ReturnActual] := fbHTTP_Values.asPropertyValue[_Domoticz_eHTTP_PropertyNames.UsageDelivery]; 
		END_IF
		
	//General / other
	ELSIF fbHTTP_Values.axMatchFound[_Domoticz_eHTTP_PropertyNames.ObjectType] 
	AND fbHTTP_Values.asPropertyValue[_Domoticz_eHTTP_PropertyNames.ObjectType] = Domoticz_Constants.sType_General THEN
		
		//SubType is available, but not used
		//If usage type found, subtype is presumably kWh or Gas > Electric (counter+instant)
		//Differs from P1, because otherwise MQTT messages are also off (they come in only at 1 and 2)
		IF fbHTTP_Values.axMatchFound[_Domoticz_eHTTP_PropertyNames.Usage] THEN
			xHTTP_TypeMatched := TRUE;
			IF fbHTTP_Values.axMatchFound[_Domoticz_eHTTP_PropertyNames.Usage] THEN 	//Usage
				scObjectData.asValue[Domoticz_eSValues_Usage.Usage] := fbHTTP_Values.asPropertyValue[_Domoticz_eHTTP_PropertyNames.Usage]; 
			END_IF
			IF fbHTTP_Values.axMatchFound[_Domoticz_eHTTP_PropertyNames.Counter] THEN 	//Counter
				scObjectData.asValue[Domoticz_eSValues_Usage.UsageCumulative] := fbHTTP_Values.asPropertyValue[_Domoticz_eHTTP_PropertyNames.Counter]; 
			ELSIF fbHTTP_Values.axMatchFound[_Domoticz_eHTTP_PropertyNames.Data] THEN 	//Counter
				scObjectData.asValue[Domoticz_eSValues_Usage.UsageCumulative] := fbHTTP_Values.asPropertyValue[_Domoticz_eHTTP_PropertyNames.Data]; 
			END_IF
			IF fbHTTP_Values.axMatchFound[_Domoticz_eHTTP_PropertyNames.CounterToday] THEN //Usage today
				scObjectData.asValue[Domoticz_eSValues_Usage.UsageToday] := fbHTTP_Values.asPropertyValue[_Domoticz_eHTTP_PropertyNames.CounterToday]; 
			END_IF
		//Other general types
		ELSE
			xHTTP_TypeMatched := FALSE;
			IF fbHTTP_Values.axMatchFound[_Domoticz_eHTTP_PropertyNames.Data] THEN 
				scObjectData.asValue[Domoticz_eSValues_General.General] := fbHTTP_Values.asPropertyValue[_Domoticz_eHTTP_PropertyNames.Data];
			END_IF	//Data
		END_IF
		
	//Other type > just pass data
	ELSIF fbHTTP_Values.axMatchFound[_Domoticz_eHTTP_PropertyNames.ObjectType] THEN
		xHTTP_TypeMatched := FALSE;
		IF fbHTTP_Values.axMatchFound[_Domoticz_eHTTP_PropertyNames.Data] THEN 
			scObjectData.asValue[Domoticz_eSValues_General.General] := fbHTTP_Values.asPropertyValue[_Domoticz_eHTTP_PropertyNames.Data]; 
		END_IF	//Data
				
	//No type available
	ELSIF NOT fbHTTP_Values.axMatchFound[_Domoticz_eHTTP_PropertyNames.ObjectType] THEN
		xHTTP_DataError := TRUE;
	END_IF

	//Add last update
	IF fbHTTP_Values.axMatchFound[_Domoticz_eHTTP_PropertyNames.LastUpdate] THEN
		scObjectData.dtLastUpdate := fbHTTP_Values.adtPropertyValue[_Domoticz_eHTTP_PropertyNames.LastUpdate];
	ELSE
		scObjectData.dtLastUpdate := DT#1970-1-1-0:0:0;
	END_IF
	
	//Convert data so it has max. two decimals at the end
	IF xHTTP_TypeMatched THEN
		FOR wX := 1 TO Domoticz_Constants.uiMaxSValues DO
			IF scObjectData.asValue[wX] <> '' THEN
				scObjectData.asValue[wX] := TO_STRING(_Domoticz_RoundDecimals(TO_REAL(scObjectData.asValue[wX]),2));
			END_IF
		END_FOR		
	END_IF
			
	//Add info
	scObjectData.sDeviceType := fbHTTP_Values.asPropertyValue[_Domoticz_eHTTP_PropertyNames.ObjectType];	//Transfer type
	scObjectData.dtTimeStamp := dtTimeStamp;	//Add timestamp
	scObjectData.eSource := _Domoticz_eDataSource.HTTP;	//Source is HTTP
	
END_IF
END_ACTION

END_FUNCTION_BLOCK

// Functions/_Domoticz_StringExtractColor
{attribute 'conditionalshow_all_locals'}
{attribute 'conditionalshow'}
FUNCTION _Domoticz_StringExtractColor :STRING(Domoticz_Constants.uiMaxSValuesize)
VAR_INPUT
	sData		:STRING(Domoticz_Constants.uiMaxSValuesize);
	eColor		:Domoticz_eSValues_Colors;
END_VAR
VAR
	//Data processing
	psData		:POINTER TO STRING(Domoticz_Constants.uiMaxSValuesize);
	sSearch		:STRING(2);
	psSearch	:POINTER TO STRING(2);
	sExtract	:STRING(3);
	psExtract	:POINTER TO STRING(4);		//255 + Closing
	
	//Positions
	iPosColor	:INT;
	iPosColom	:INT;
	iPosComma	:INT;
	iPosAccolade:INT;
END_VAR

//Format:
//{\"b\":84,\"cw\":0,\"g\":188,\"m\":3,\"r\":254,\"t\":0,\"ww\":0}

IF eColor >= Domoticz_eSValues_Colors.Red AND eColor <= TO_INT(Domoticz_eSValues_Colors.WarmWhite)
AND sData <> '' THEN

	psData := ADR(sData);
	psSearch := ADR(sSearch);
	psExtract := ADR(sExtract);
	
	//Find position of text
	sSearch := Domoticz_Constants.asProperty_Colors[eColor];
	iPosColor := StrFindA(psData, psSearch, TO_UINT(0));	//Find pos of text
	
	//Find position of colom
	sSearch := ':';
	iPosColom := StrFindA(psData, psSearch, TO_UINT(iPosColor));	//Find pos of colom
	
	//Find position of comma
	sSearch := ',';
	iPosComma := StrFindA(psData, psSearch, TO_UINT(iPosColom));	//Find pos of comma
	
	//Find position of accolade
	sSearch := '}';
	iPosAccolade := StrFindA(psData, psSearch, TO_UINT(iPosColom));	//Find pos of accolade
	
	//Extract data
	//Comma present
	IF iPosComma > 0 THEN
		StrMidA(psData, Domoticz_Constants.uiMaxSValuesize, (iPosComma-iPosColom-1), iPosColom+1,  psExtract, 4);
	//Accolade present
	ELSIF iPosAccolade > 0 THEN
		StrMidA(psData, Domoticz_Constants.uiMaxSValuesize, (iPosAccolade-iPosColom-1), iPosColom+1,  psExtract, 4);
	//Extract last bit
	ELSE
		StrMidA(psData, Domoticz_Constants.uiMaxSValuesize, TO_INT(StrLenA(psData)-iPosColom-1), iPosColom+1,  psExtract, 4);
	END_IF
	StrTrimA(psExtract);
	
	//Output
	_Domoticz_StringExtractColor := sExtract;
	
ELSE
	_Domoticz_StringExtractColor := '';
END_IF

END_FUNCTION

// Functions/_Domoticz_StringExtractAfterDot
{attribute 'conditionalshow_all_locals'}
{attribute 'conditionalshow'}
FUNCTION _Domoticz_StringExtractAfterDot :STRING(Domoticz_Constants.uiInstanceName);
VAR_INPUT
	sData		:STRING(Domoticz_Constants.uiInstanceName);
END_VAR
VAR
	psData		:POINTER TO STRING(Domoticz_Constants.uiInstanceName);
	sFind		:STRING(Domoticz_Constants.uiInstanceName);	
	psFind		:POINTER TO STRING(Domoticz_Constants.uiInstanceName);
	sExtract	:STRING(Domoticz_Constants.uiInstanceName);	
	psExtract	:POINTER TO STRING(Domoticz_Constants.uiInstanceName);	
	
	byDotLoop	:BYTE;
	uiFindDot	:UINT;
	uiLastDot	:UINT;
END_VAR

IF sData <> '' THEN
	//Load pointers
	psData := ADR(sData);
	psFind := ADR(sFind);
	psExtract := ADR(sExtract);
	
	
	sFind := '.';
	uiFindDot := 0;
	//Find positions of all possible dots
	FOR byDotLoop := 0 TO 15 DO
		uiFindDot := TO_UINT(StrFindA(psData ,psFind, uiFindDot+1)); 
		IF uiFindDot > 0 THEN
			uiLastDot := uiFindDot;
		END_IF
	END_FOR
		
	//Check data
	IF uiLastDot > 0 THEN
		StrMidA(psData, Domoticz_Constants.uiInstanceName, TO_INT(StrLenA(psData)-uiLastDot), TO_INT(uiLastDot+1), psExtract, Domoticz_Constants.uiInstanceName);
	ELSE
		sExtract := sData;
	END_IF
	
	//Convert
	_Domoticz_StringExtractAfterDot := sExtract;
	
ELSE
	_Domoticz_StringExtractAfterDot := '';
END_IF

END_FUNCTION

// Function Blocks/Objects/_Domoticz_ObjectInt_InOut
{attribute 'conditionalshow'}
FUNCTION_BLOCK _Domoticz_ObjectInt_InOut EXTENDS _Domoticz_ObjectInt_Out
VAR_INPUT
	iValueSet					:INT;
END_VAR
VAR
	xUseOnlyNValue_int			:BOOL;
END_VAR

IF __ISVALIDREF(scConnector) THEN
	Main();
END_IF

ACTION Main:
{attribute 'conditionalshow'}
//Process main function
SUPER^.Main(scConnector:=scConnector);

//Transfer data to input
IF iValueSet = iValueSetLimitLow_int THEN
	iValue_In 	:= 0;
	asValue_In[1]:= '';	//Not used
ELSIF iValueSet = iValueSetLimitHigh_int THEN
	iValue_In 	:= 1;
	asValue_In[1]:= '';	//Not used
ELSE
	IF NOT xUseOnlyNValue_int THEN
		iValue_In 	:= 2;		//2 means sValue is used
		asValue_In[1]:= TO_STRING(iValueSet);
	ELSIF xUseOnlyNValue_int THEN
		iValue_In := iValueSet;
	END_IF
END_IF
END_ACTION

{attribute 'monitoring' := 'call'} PROPERTY xUseOnlyNValue :BOOL
SET
xUseOnlyNValue_int := xUseOnlyNValue;
END_SET
GET
xUseOnlyNValue := xUseOnlyNValue_int;
END_GET
END_PROPERTY

END_FUNCTION_BLOCK

// Function Blocks/Objects/_Domoticz_ObjectInt_Out
{attribute 'conditionalshow'}
FUNCTION_BLOCK _Domoticz_ObjectInt_Out EXTENDS _Domoticz_Object
VAR_INPUT
END_VAR
VAR_OUTPUT
	iValueAct					:INT;
END_VAR
VAR
	iValueSetLimitLow_int		:INT := 0;
	iValueSetLimitHigh_int		:INT := 100;
END_VAR

IF __ISVALIDREF(scConnector) THEN
	Main();
END_IF

ACTION Main:
{attribute 'conditionalshow'}
//Process main function
SUPER^.Main(scConnector:=scConnector);

//Transfer data to output
IF uiIdentifier_int > 0 AND xUpdateReceived_int THEN 
	IF (iValue_Out >= iValueSetLimitLow_int OR iValue_Out <= iValueSetLimitHigh_int)
	AND iValue_Out <> 2 THEN		//2 means that asValue is used (normally)
		iValueAct := iValue_Out;
	ELSE
		IF asValue_Out[1] <> '' THEN //Valid
			iValueAct := TO_INT(asValue_Out[1]);
		END_IF
	END_IF
ELSIF uiIdentifier_int = 0 THEN 
	iValueAct := 0; 
END_IF
END_ACTION

{attribute 'monitoring' := 'call'} PROPERTY iValueSetLimitLow :INT
SET
iValueSetLimitLow_int := iValueSetLimitLow;
END_SET
GET
iValueSetLimitLow := iValueSetLimitLow_int;
END_GET
END_PROPERTY

{attribute 'monitoring' := 'call'} PROPERTY iValueSetLimitHigh :INT
SET
iValueSetLimitHigh_int := iValueSetLimitHigh;
END_SET
GET
iValueSetLimitHigh := iValueSetLimitHigh_int;
END_GET
END_PROPERTY

END_FUNCTION_BLOCK

// Function Blocks/Objects/_Domoticz_ObjectString_InOut
{attribute 'conditionalshow'}
FUNCTION_BLOCK _Domoticz_ObjectString_InOut EXTENDS _Domoticz_ObjectString_Out
VAR_INPUT
	sValueSet					:STRING(Domoticz_Constants.uiMaxSValuesize);
END_VAR
VAR
END_VAR

IF __ISVALIDREF(scConnector) THEN
	Main();
END_IF

ACTION Main:
{attribute 'conditionalshow'}
//Process main function
SUPER^.Main(scConnector:=scConnector);

//Transfer data to input
asValue_In[1] := sValueSet;
END_ACTION

END_FUNCTION_BLOCK

// Function Blocks/Hardware/System/Network/Domoticz_SystemAliveChecker
{attribute 'conditionalshow_all_locals'}
FUNCTION_BLOCK Domoticz_SystemAliveChecker EXTENDS _Domoticz_Connector_Out
VAR_INPUT
	uiIdentifier				:UINT;	//Device to ping
END_VAR
VAR_OUTPUT
	xAlive						:BOOL;
END_VAR
VAR
	afb_ObjectBool_Out			:ARRAY[1..1] OF _Domoticz_ObjectBool_Out;
END_VAR

IF __ISVALIDREF(scConnector) THEN
	Main();
END_IF

ACTION Main:
{attribute 'conditionalshow'}
//Call parent function
SUPER^.Main();

//Call all functions
//Data timeout is only updated when device changes status so likely will be disabled
afb_ObjectBool_Out[1].tDataTimeOut := T#12H;
afb_ObjectBool_Out[1](scConnector := scConnector,	uiIdentifier := uiIdentifier, 	xValueAct => xAlive);

//Errors
fbEI_DataTimeOut.sInstanceName := sInstanceName;
fbEI_DataTimeOut.tErrorDelay := T#500MS;	//Give objects TIME TO be overruled BY other updates
fbEI_DataTimeOut(
	scConnector:= scConnector,
	xError:= xDataTimeOut_int
			AND (afb_ObjectBool_Out[1].xDataTimedOut),
	eErrorID:= Domoticz_eErrors.ObjectDataTimeOut
);
END_ACTION

END_FUNCTION_BLOCK

// Function Blocks/Hardware/System/Network/Domoticz_MotherboardSensors
{attribute 'conditionalshow_all_locals'}
FUNCTION_BLOCK Domoticz_MotherboardSensors EXTENDS _Domoticz_Connector_Out
VAR_INPUT
	uiIdentifier_CPU			:UINT;	//CPU Usage
	uiIdentifier_Memory			:UINT;	//Memory Usage
	uiIdentifier_Process		:UINT;	//Process Usage
	uiIdentifier_HDD			:UINT;	//HDD
	uiIdentifier_Temperature	:UINT;	//CPU Temperature
END_VAR
VAR_OUTPUT
	rCPU						:REAL;
	rMemory						:REAL;
	rProcess					:REAL;
	rHDD						:REAL;
	rTemperature				:REAL;
END_VAR
VAR
	afb_ObjectReal_Out			:ARRAY[1..5] OF _Domoticz_ObjectReal_Out;
	
	rThresholdCPUHigh_int		:REAL := 75;
	fbSP_CPUHigh				:_Domoticz_SwitchPoint;
	fbEI_CPUHigh				:Domoticz_ErrorInterface;
	rThresholdCPUMax_int		:REAL := 95;
	fbSP_CPUMax					:_Domoticz_SwitchPoint;
	fbEI_CPUMax					:Domoticz_ErrorInterface;
	rThresholdMemoryHigh_int	:REAL := 75;
	fbSP_MemoryHigh				:_Domoticz_SwitchPoint;
	fbEI_MemoryHigh				:Domoticz_ErrorInterface;
	rThresholdMemoryMax_int		:REAL := 95;
	fbSP_MemoryMax				:_Domoticz_SwitchPoint;
	fbEI_MemoryMax				:Domoticz_ErrorInterface;
	rThresholdHDDHigh_int		:REAL := 75;
	fbSP_HDDHigh				:_Domoticz_SwitchPoint;
	fbEI_HDDHigh				:Domoticz_ErrorInterface;
	rThresholdHDDMax_int		:REAL := 95;
	fbSP_HDDMax					:_Domoticz_SwitchPoint;
	fbEI_HDDMax					:Domoticz_ErrorInterface;
	rThresholdTemperatureHigh_int:REAL := 60;
	fbSP_TemperatureHigh		:_Domoticz_SwitchPoint;
	fbEI_TemperatureHigh		:Domoticz_ErrorInterface;
	rThresholdTemperatureMax_int :REAL := 80;
	fbSP_TemperatureMax			:_Domoticz_SwitchPoint;
	fbEI_TemperatureMax			:Domoticz_ErrorInterface;
END_VAR

IF __ISVALIDREF(scConnector) THEN
	Main();
END_IF

ACTION Main:
{attribute 'conditionalshow'}
//Call parent function
SUPER^.Main();

//Call all functions
//Data timeout (update rate is every two minute or so)
afb_ObjectReal_Out[1].tDataTimeOut := T#15M;
afb_ObjectReal_Out[1](scConnector := scConnector, 	uiIdentifier := uiIdentifier_CPU, 			rxUpdateInterlock := rxUpdateInterlock_int,			rValueAct => rCPU);

afb_ObjectReal_Out[2].tDataTimeOut := T#15M;
afb_ObjectReal_Out[2](scConnector := scConnector, 	uiIdentifier := uiIdentifier_Memory, 		rxUpdateInterlock := rxUpdateInterlock_int,			rValueAct => rMemory);

afb_ObjectReal_Out[3].tDataTimeOut := T#15M;
afb_ObjectReal_Out[3](scConnector := scConnector, 	uiIdentifier := uiIdentifier_Process, 		rxUpdateInterlock := rxUpdateInterlock_int,			rValueAct => rProcess);

afb_ObjectReal_Out[4].tDataTimeOut := T#15M;
afb_ObjectReal_Out[4](scConnector := scConnector, 	uiIdentifier := uiIdentifier_HDD, 			rxUpdateInterlock := rxUpdateInterlock_int,			rValueAct => rHDD);

afb_ObjectReal_Out[5].tDataTimeOut := T#15M;
afb_ObjectReal_Out[5](scConnector := scConnector, 	uiIdentifier := uiIdentifier_Temperature, 	rxUpdateInterlock := rxUpdateInterlock_int,			rValueAct => rTemperature);								  
									  
//Errors
//********************************************DATA
fbEI_DataTimeOut.sInstanceName := sInstanceName;
fbEI_DataTimeOut.tErrorDelay := T#500MS;	//Give objects TIME TO be overruled BY other updates
fbEI_DataTimeOut(
	scConnector:= scConnector,
	xError:= xDataTimeOut_int
			AND (afb_ObjectReal_Out[1].xDataTimedOut
			OR afb_ObjectReal_Out[2].xDataTimedOut
			OR afb_ObjectReal_Out[3].xDataTimedOut
			OR afb_ObjectReal_Out[4].xDataTimedOut
			OR afb_ObjectReal_Out[5].xDataTimedOut),
	eErrorID:= Domoticz_eErrors.ObjectDataTimeOut
);

//********************************************CPU
fbSP_CPUHigh(
	xEnable:= rCPU > 0,
	rInput:= rCPU, 
	rSwitchPoint:= rThresholdCPUHigh_int, 
	rHysteresis:= 10, 
	xInvert:= FALSE, 
	xOut=> );
fbEI_CPUHigh.sInstanceName := sInstanceName;
fbEI_CPUHigh.sErrorInfo := TO_STRING(TO_INT(_Domoticz_RoundDecimals(rCPU,0)));
fbEI_CPUHigh.sErrorInfo := CONCAT(fbEI_CPUHigh.sErrorInfo, ' %');
fbEI_CPUHigh(
	scConnector:= scConnector,
	xError:= fbSP_CPUHigh.xOut 
			AND rThresholdCPUHigh_int > 0
			AND uiIdentifier_CPU > 0,
	eErrorID:= Domoticz_eErrors.Motherboard_CpuUsageHigh
);

fbSP_CPUMax(
	xEnable:= rCPU > 0,
	rInput:= rCPU, 
	rSwitchPoint:= rThresholdCPUMax_int, 
	rHysteresis:= 10, 
	xInvert:= FALSE, 
	xOut=> );
fbEI_CPUMax.sInstanceName := sInstanceName;
fbEI_CPUMax.sErrorInfo := TO_STRING(TO_INT(_Domoticz_RoundDecimals(rCPU,0)));
fbEI_CPUMax.sErrorInfo := CONCAT(fbEI_CPUMax.sErrorInfo, ' %');
fbEI_CPUMax(
	scConnector:= scConnector,
	xError:= fbSP_CPUMax.xOut
			AND rThresholdCPUMax_int > 0
			AND uiIdentifier_CPU > 0,
	eErrorID:= Domoticz_eErrors.Motherboard_CpuUsageMax
);

//********************************************MEMORY
fbSP_MemoryHigh(
	xEnable:= rMemory > 0,
	rInput:= rMemory, 
	rSwitchPoint:= rThresholdMemoryHigh_int, 
	rHysteresis:= 10, 
	xInvert:= FALSE, 
	xOut=> );
fbEI_MemoryHigh.sInstanceName := sInstanceName;
fbEI_MemoryHigh.sErrorInfo := TO_STRING(TO_INT(_Domoticz_RoundDecimals(rMemory,0)));
fbEI_MemoryHigh.sErrorInfo := CONCAT(fbEI_MemoryHigh.sErrorInfo, ' %');
fbEI_MemoryHigh(
	scConnector:= scConnector,
	xError:= fbSP_MemoryHigh.xOut
			AND rThresholdMemoryHigh_int > 0
			AND uiIdentifier_Memory > 0,
	eErrorID:= Domoticz_eErrors.Motherboard_MemoryUsageHigh
);

fbSP_MemoryMax(
	xEnable:= rMemory > 0,
	rInput:= rMemory, 
	rSwitchPoint:= rThresholdMemoryMax_int, 
	rHysteresis:= 10, 
	xInvert:= FALSE, 
	xOut=> );
fbEI_MemoryMax.sInstanceName := sInstanceName;
fbEI_MemoryMax.sErrorInfo := TO_STRING(TO_INT(_Domoticz_RoundDecimals(rMemory,0)));
fbEI_MemoryMax.sErrorInfo := CONCAT(fbEI_MemoryMax.sErrorInfo, ' %');
fbEI_MemoryMax(
	scConnector:= scConnector,
	xError:= fbSP_MemoryMax.xOut 
			AND rThresholdMemoryMax_int > 0
			AND uiIdentifier_Memory > 0,
	eErrorID:= Domoticz_eErrors.Motherboard_MemoryUsageMax
);

//********************************************HDD
fbSP_HDDHigh(
	xEnable:= rHDD > 0,
	rInput:= rHDD, 
	rSwitchPoint:= rThresholdHDDHigh_int, 
	rHysteresis:= 5, 
	xInvert:= FALSE, 
	xOut=> );
fbEI_HDDHigh.sInstanceName := sInstanceName;
fbEI_HDDHigh.sErrorInfo := TO_STRING(TO_INT(_Domoticz_RoundDecimals(rHDD,0)));
fbEI_HDDHigh.sErrorInfo := CONCAT(fbEI_HDDHigh.sErrorInfo, ' %');
fbEI_HDDHigh(
	scConnector:= scConnector,
	xError:= fbSP_HDDHigh.xOut 
			AND rThresholdHDDHigh_int > 0 
			AND uiIdentifier_HDD > 0,
	eErrorID:= Domoticz_eErrors.Motherboard_HDDUsageHigh
);

fbSP_HDDMax(
	xEnable:= rHDD > 0,
	rInput:= rHDD, 
	rSwitchPoint:= rThresholdHDDMax_int, 
	rHysteresis:= 5, 
	xInvert:= FALSE, 
	xOut=> );
fbEI_HDDMax.sInstanceName := sInstanceName;
fbEI_HDDMax.sErrorInfo := TO_STRING(TO_INT(_Domoticz_RoundDecimals(rHDD,0)));
fbEI_HDDMax.sErrorInfo := CONCAT(fbEI_HDDMax.sErrorInfo, ' %');
fbEI_HDDMax(
	scConnector:= scConnector,
	xError:= fbSP_HDDMax.xOut 
			AND rThresholdHDDMax_int > 0
			AND uiIdentifier_HDD > 0,
	eErrorID:= Domoticz_eErrors.Motherboard_HDDUsageMax
);

//********************************************TEMPERATURE
fbSP_TemperatureHigh(
	xEnable:= rTemperature > 0,
	rInput:= rTemperature, 
	rSwitchPoint:= rThresholdTemperatureHigh_int, 
	rHysteresis:= 5, 
	xInvert:= FALSE, 
	xOut=> );
fbEI_TemperatureHigh.sInstanceName := sInstanceName;
fbEI_TemperatureHigh.sErrorInfo := TO_STRING(_Domoticz_RoundDecimals(rTemperature,1));
fbEI_TemperatureHigh.sErrorInfo := CONCAT(fbEI_TemperatureHigh.sErrorInfo, ' C');
fbEI_TemperatureHigh(
	scConnector:= scConnector,
	xError:= fbSP_TemperatureHigh.xOut 
			AND rThresholdTemperatureHigh_int > 0
			AND uiIdentifier_Temperature > 0,
	eErrorID:= Domoticz_eErrors.Motherboard_TemperatureHigh
);

fbSP_TemperatureMax(
	xEnable:= rTemperature > 0,
	rInput:= rTemperature, 
	rSwitchPoint:= rThresholdTemperatureMax_int, 
	rHysteresis:= 5, 
	xInvert:= FALSE, 
	xOut=> );
fbEI_TemperatureMax.sInstanceName := sInstanceName;
fbEI_TemperatureMax.sErrorInfo := TO_STRING(_Domoticz_RoundDecimals(rTemperature,1));
fbEI_TemperatureMax.sErrorInfo := CONCAT(fbEI_TemperatureMax.sErrorInfo, ' C');
fbEI_TemperatureMax(
	scConnector:= scConnector,
	xError:= fbSP_TemperatureMax.xOut 
			AND rThresholdTemperatureMax_int > 0
			AND uiIdentifier_Temperature > 0,
	eErrorID:= Domoticz_eErrors.Motherboard_TemperatureMax
);
END_ACTION

{attribute 'monitoring' := 'call'} PROPERTY rThresholdCPUHigh :REAL
SET
rThresholdCPUHigh_int := rThresholdCPUHigh;
END_SET
GET
rThresholdCPUHigh := rThresholdCPUHigh_int;
END_GET
END_PROPERTY

{attribute 'monitoring' := 'call'} PROPERTY rThresholdCPUMax :REAL
SET
rThresholdCPUMax_int := rThresholdCPUMax;
END_SET
GET
rThresholdCPUMax := rThresholdCPUMax_int;
END_GET
END_PROPERTY

{attribute 'monitoring' := 'call'} PROPERTY rThresholdMemoryHigh :REAL
SET
rThresholdMemoryHigh_int := rThresholdMemoryHigh;
END_SET
GET
rThresholdMemoryHigh := rThresholdMemoryHigh_int;
END_GET
END_PROPERTY

{attribute 'monitoring' := 'call'} PROPERTY rThresholdMemoryMax :REAL
SET
rThresholdMemoryMax_int := rThresholdMemoryMax;
END_SET
GET
rThresholdMemoryMax := rThresholdMemoryMax_int;
END_GET
END_PROPERTY

{attribute 'monitoring' := 'call'} PROPERTY rThresholdHDDHigh :REAL
SET
rThresholdHDDHigh_int := rThresholdHDDHigh;
END_SET
GET
rThresholdHDDHigh := rThresholdHDDHigh_int;
END_GET
END_PROPERTY

{attribute 'monitoring' := 'call'} PROPERTY rThresholdHDDMax :REAL
SET
rThresholdHDDMax_int := rThresholdHDDMax;
END_SET
GET
rThresholdHDDMax := rThresholdHDDMax_int;
END_GET
END_PROPERTY

{attribute 'monitoring' := 'call'} PROPERTY rThresholdTemperatureHigh :REAL
SET
rThresholdTemperatureHigh_int := rThresholdTemperatureHigh;
END_SET
GET
rThresholdTemperatureHigh := rThresholdTemperatureHigh_int;
END_GET
END_PROPERTY

{attribute 'monitoring' := 'call'} PROPERTY rThresholdTemperatureMax :REAL
SET
rThresholdTemperatureMax_int := rThresholdTemperatureMax;
END_SET
GET
rThresholdTemperatureMax := rThresholdTemperatureMax_int;
END_GET
END_PROPERTY

END_FUNCTION_BLOCK

// Function Blocks/Hardware/System/Network/Domoticz_UPSMonitor
{attribute 'conditionalshow_all_locals'}
FUNCTION_BLOCK Domoticz_UPSMonitor EXTENDS _Domoticz_Connector_Out
VAR_INPUT
	uiIdentifier_MainsVoltage	:UINT;
	uiIdentifier_MainsFrequency	:UINT;
	uiIdentifier_ChargeLevel	:UINT;
	uiIdentifier_LoadLevel		:UINT;
	uiIdentifier_BackupTime		:UINT;
	uiIdentifier_Status			:UINT;
END_VAR
VAR_OUTPUT
	rMainsVoltage				:REAL;
	rMainsFrequency				:REAL;
	rChargeLevel				:REAL;
	rLoadLevel					:REAL;
	tBackupTime					:TIME;
	sStatus						:STRING(Domoticz_Constants.uiMaxSValuesize);
END_VAR
VAR
	afb_ObjectReal_Out			:ARRAY[1..5] OF _Domoticz_ObjectReal_Out;
	afb_ObjectString_Out		:ARRAY[1..1] OF _Domoticz_ObjectString_Out;
	
	rThresholdVoltage_int		:REAL := 200;
	rThresholdFrequency_int		:REAL := 50;
	fbEI_PowerFailure			:Domoticz_ErrorInterface;
	
	rThresholdChargeLevelLow_int:REAL := 50;	//%
	fbSP_ChargeLevelLow			:_Domoticz_SwitchPoint;
	fbEI_ChargeLevelLow			:Domoticz_ErrorInterface;
	
	rThresholdChargeLevelCritical_int:REAL := 25;	//%
	fbSP_ChargeLevelCritical	:_Domoticz_SwitchPoint;
	fbEI_ChargeLevelCritical	:Domoticz_ErrorInterface;
	
	rThresholdLoadLevelHigh_int	:REAL := 75;	//%
	fbSP_LoadLevelHigh			:_Domoticz_SwitchPoint;
	fbEI_LoadLevelHigh			:Domoticz_ErrorInterface;
	
	rThresholdLoadLevelMax_int	:REAL := 95;	//%
	fbSP_LoadLevelMax			:_Domoticz_SwitchPoint;
	fbEI_LoadLevelMax			:Domoticz_ErrorInterface;

	fbEI_BackUpTime_5min		:Domoticz_ErrorInterface;
	fbEI_BackUpTime_1min		:Domoticz_ErrorInterface;

END_VAR

IF __ISVALIDREF(scConnector) THEN
	Main();
END_IF

ACTION Main:
{attribute 'conditionalshow'}
//Call parent function
SUPER^.Main();

//Call all functions
//Data timeout (update rate is every two minute or so)
afb_ObjectReal_Out[1].tDataTimeOut := T#15M;
afb_ObjectReal_Out[1](	scConnector := scConnector, 	uiIdentifier := uiIdentifier_MainsVoltage, 		rxUpdateInterlock := rxUpdateInterlock_int,			rValueAct => rMainsVoltage);

afb_ObjectReal_Out[2].tDataTimeOut := T#15M;
afb_ObjectReal_Out[2](	scConnector := scConnector, 	uiIdentifier := uiIdentifier_MainsFrequency, 	rxUpdateInterlock := rxUpdateInterlock_int,			rValueAct => rMainsFrequency);

afb_ObjectReal_Out[3].tDataTimeOut := T#15M;
afb_ObjectReal_Out[3].eDataSource := _Domoticz_eDataSource.HTTP;
afb_ObjectReal_Out[3](	scConnector := scConnector, 	uiIdentifier := uiIdentifier_ChargeLevel, 		rxUpdateInterlock := rxUpdateInterlock_int,			rValueAct => rChargeLevel);
                                                                                                                                                                                  
afb_ObjectReal_Out[4].tDataTimeOut := T#15M;         
afb_ObjectReal_Out[4].eDataSource := _Domoticz_eDataSource.HTTP;                                                                                                                             
afb_ObjectReal_Out[4](	scConnector := scConnector, 	uiIdentifier := uiIdentifier_LoadLevel, 		rxUpdateInterlock := rxUpdateInterlock_int,			rValueAct => rLoadLevel);
                                                                                                                                                                                  
afb_ObjectReal_Out[5].tDataTimeOut := T#15M;                                                                                                                                    
afb_ObjectReal_Out[5].rScalingAct := 1000;  
afb_ObjectReal_Out[5].eDataSource := _Domoticz_eDataSource.HTTP;
afb_ObjectReal_Out[5](	scConnector := scConnector, 	uiIdentifier := uiIdentifier_BackupTime,		rxUpdateInterlock := rxUpdateInterlock_int);	
                                                                                                                                                                                  
afb_ObjectString_Out[1].tDataTimeOut := T#15M;
afb_ObjectString_Out[1].eDataSource := _Domoticz_eDataSource.HTTP;                                                                                                                                  
afb_ObjectString_Out[1](scConnector := scConnector, 	uiIdentifier := uiIdentifier_Status, 			rxUpdateInterlock := rxUpdateInterlock_int,			sValueAct => sStatus);

//Output transformation
tBackupTime := TO_TIME(afb_ObjectReal_Out[5].rValueAct);									  

//Errors
//********************************************DATA
fbEI_DataTimeOut.sInstanceName := sInstanceName;
fbEI_DataTimeOut.tErrorDelay := T#500MS;	//Give objects TIME TO be overruled BY other updates
fbEI_DataTimeOut(
	scConnector:= scConnector,
	xError:= xDataTimeOut_int
			AND (afb_ObjectReal_Out[1].xDataTimedOut
			OR afb_ObjectReal_Out[2].xDataTimedOut
			OR afb_ObjectReal_Out[3].xDataTimedOut
			OR afb_ObjectReal_Out[4].xDataTimedOut
			OR afb_ObjectReal_Out[5].xDataTimedOut
			OR afb_ObjectString_Out[1].xDataTimedOut),
	eErrorID:= Domoticz_eErrors.ObjectDataTimeOut
);

//********************************************POWER FAILURE
fbEI_PowerFailure.sInstanceName := sInstanceName;
fbEI_PowerFailure.sErrorInfo := TO_STRING(TO_INT(_Domoticz_RoundDecimals(rMainsVoltage,0)));
fbEI_PowerFailure.sErrorInfo := CONCAT(fbEI_PowerFailure.sErrorInfo, ' V / ');
fbEI_PowerFailure.sErrorInfo := CONCAT(fbEI_PowerFailure.sErrorInfo, TO_STRING(TO_INT(_Domoticz_RoundDecimals(rMainsFrequency,0))));
fbEI_PowerFailure.sErrorInfo := CONCAT(fbEI_PowerFailure.sErrorInfo, ' Hz');
fbEI_PowerFailure(
	scConnector:= scConnector,
	xError:= scConnector.xServerConnected
			AND ((rMainsVoltage < rThresholdVoltage_int AND uiIdentifier_MainsVoltage > 0)
			OR ((rMainsFrequency < (rThresholdFrequency_int - 5) OR rMainsFrequency > (rThresholdFrequency_int + 5)) AND uiIdentifier_MainsFrequency > 0)),
	eErrorID:= Domoticz_eErrors.UPS_PowerFailure
);

//********************************************CHARGE LEVEL
fbSP_ChargeLevelLow(
	xEnable:= rChargeLevel > 0,
	rInput:= rChargeLevel, 
	rSwitchPoint:= rThresholdChargeLevelLow_int, 
	rHysteresis:= 5, 
	xInvert:= TRUE, 
	xOut=> );
fbEI_ChargeLevelLow.sInstanceName := sInstanceName;
fbEI_ChargeLevelLow.sErrorInfo := TO_STRING(TO_INT(_Domoticz_RoundDecimals(rChargeLevel,0)));
fbEI_ChargeLevelLow.sErrorInfo := CONCAT(fbEI_ChargeLevelLow.sErrorInfo, ' %');
fbEI_ChargeLevelLow(
	scConnector:= scConnector,
	xError:= fbSP_ChargeLevelLow.xOut
			AND rThresholdChargeLevelLow_int > 0
			AND uiIdentifier_ChargeLevel > 0,
	eErrorID:= Domoticz_eErrors.UPS_ChargeLevelLow
);

fbSP_ChargeLevelCritical(
	xEnable:= rChargeLevel > 0,
	rInput:= rChargeLevel, 
	rSwitchPoint:= rThresholdChargeLevelCritical_int, 
	rHysteresis:= 5, 
	xInvert:= TRUE, 
	xOut=> );
fbEI_ChargeLevelCritical.sInstanceName := sInstanceName;
fbEI_ChargeLevelCritical.sErrorInfo := TO_STRING(TO_INT(_Domoticz_RoundDecimals(rChargeLevel,0)));
fbEI_ChargeLevelCritical.sErrorInfo := CONCAT(fbEI_ChargeLevelCritical.sErrorInfo, ' %');
fbEI_ChargeLevelCritical(
	scConnector:= scConnector,
	xError:= fbSP_ChargeLevelCritical.xOut 
			AND rThresholdChargeLevelCritical_int > 0
			AND uiIdentifier_ChargeLevel > 0,
	eErrorID:= Domoticz_eErrors.UPS_ChargeLevelCritical
);

//********************************************LOAD LEVEL
fbSP_LoadLevelHigh(
	xEnable:= rLoadLevel > 0,
	rInput:= rLoadLevel, 
	rSwitchPoint:= rThresholdLoadLevelHigh_int, 
	rHysteresis:= 5, 
	xInvert:= FALSE, 
	xOut=> );
fbEI_LoadLevelHigh.sInstanceName := sInstanceName;
fbEI_LoadLevelHigh.sErrorInfo := TO_STRING(TO_INT(_Domoticz_RoundDecimals(rLoadLevel,0)));
fbEI_LoadLevelHigh.sErrorInfo := CONCAT(fbEI_LoadLevelHigh.sErrorInfo, ' %');
fbEI_LoadLevelHigh(
	scConnector:= scConnector,
	xError:= fbSP_LoadLevelHigh.xOut 
			AND rThresholdLoadLevelHigh_int > 0
			AND uiIdentifier_LoadLevel > 0,
	eErrorID:= Domoticz_eErrors.UPS_LoadLevelHigh
);

fbSP_LoadLevelMax(
	xEnable:= rLoadLevel > 0,
	rInput:= rLoadLevel, 
	rSwitchPoint:= rThresholdLoadLevelMax_int, 
	rHysteresis:= 5, 
	xInvert:= FALSE, 
	xOut=> );
fbEI_LoadLevelMax.sInstanceName := sInstanceName;
fbEI_LoadLevelMax.sErrorInfo := TO_STRING(TO_INT(_Domoticz_RoundDecimals(rLoadLevel,0)));
fbEI_LoadLevelMax.sErrorInfo := CONCAT(fbEI_LoadLevelMax.sErrorInfo, ' %');
fbEI_LoadLevelMax(
	scConnector:= scConnector,
	xError:= fbSP_LoadLevelMax.xOut
			AND rThresholdLoadLevelMax_int > 0
			AND uiIdentifier_LoadLevel > 0,
	eErrorID:= Domoticz_eErrors.UPS_LoadLevelMax
);

//********************************************BACKUP TIME
fbEI_BackUpTime_5min.sInstanceName := sInstanceName;
fbEI_BackUpTime_5min(
	scConnector:= scConnector,
	xError:= tBackupTime > T#0MS
			AND tBackupTime < T#5M
			AND uiIdentifier_BackupTime > 0,
	eErrorID:= Domoticz_eErrors.UPS_BackupTime_5Min
);

fbEI_BackUpTime_1min.sInstanceName := sInstanceName;
fbEI_BackUpTime_1min(
	scConnector:= scConnector,
	xError:= tBackupTime > T#0MS
			AND tBackupTime < T#1M
			AND uiIdentifier_BackupTime > 0,
	eErrorID:= Domoticz_eErrors.UPS_BackupTime_1Min
);
END_ACTION

{attribute 'monitoring' := 'call'} PROPERTY rThresholdChargeLevelLow :REAL
SET
rThresholdChargeLevelLow_int := rThresholdChargeLevelLow;
END_SET
GET
rThresholdChargeLevelLow := rThresholdChargeLevelLow_int;
END_GET
END_PROPERTY

{attribute 'monitoring' := 'call'} PROPERTY rThresholdChargeLevelCritical :REAL
SET
rThresholdChargeLevelCritical_int := rThresholdChargeLevelCritical;
END_SET
GET
rThresholdChargeLevelCritical := rThresholdChargeLevelCritical_int;
END_GET
END_PROPERTY

{attribute 'monitoring' := 'call'} PROPERTY rThresholdLoadLevelHigh :REAL
SET
rThresholdLoadLevelHigh_int := rThresholdLoadLevelHigh;
END_SET
GET
rThresholdLoadLevelHigh := rThresholdLoadLevelHigh_int;
END_GET
END_PROPERTY

{attribute 'monitoring' := 'call'} PROPERTY rThresholdLoadLevelMax :REAL
SET
rThresholdLoadLevelMax_int := rThresholdLoadLevelMax;
END_SET
GET
rThresholdLoadLevelMax := rThresholdLoadLevelMax_int;
END_GET
END_PROPERTY

PROPERTY rThresholdFrequency : REAL
SET
rThresholdFrequency_int := rThresholdFrequency;
END_SET
GET
rThresholdFrequency := rThresholdFrequency_int;
END_GET
END_PROPERTY

PROPERTY rThresholdVoltage : REAL
SET
rThresholdVoltage_int := rThresholdVoltage;
END_SET
GET
rThresholdVoltage := rThresholdVoltage_int;
END_GET
END_PROPERTY

END_FUNCTION_BLOCK

// Function Blocks/Hardware/Devices/Domoticz_MiFlora
{attribute 'conditionalshow_all_locals'}
FUNCTION_BLOCK Domoticz_MiFlora EXTENDS _Domoticz_Connector_Out
VAR_INPUT
	uiIdentifier_Temperature	:UINT;	//Temperature
	uiIdentifier_Moisture		:UINT;	//Soil moisture in Cb
	uiIdentifier_Light			:UINT;	//Light intensity in Lux
	uiIdentifier_Fertility		:UINT;	//Fertility of the soil
	uiIdentifier_UpdateSwitch	:UINT;	//Switch to activate plugin update (use additional created switch per plant!)
	tUpdateRate					:TIME := T#60M;	//Limited to 1m minimal
END_VAR
VAR_OUTPUT
	rTemperature				:REAL;
	rMoisture					:REAL;
	rLux						:REAL;
	rFertility					:REAL;
END_VAR
VAR
	afb_ObjectReal_Out			:ARRAY[1..4] OF _Domoticz_ObjectReal_Out;
	afb_ObjectBool_InOut		:ARRAY[1..1] OF _Domoticz_ObjectBool_InOut;
	TON_Update					:TON;
	xTONUpdate					:BOOL;
	
	rThresholdMoistureLow_int	:REAL := 50;
	fbSP_MoistureLow			:_Domoticz_SwitchPoint;
	fbEI_MoistureLow			:Domoticz_ErrorInterface;
	
	rThresholdFertilityLow_int	:REAL := 500;
	fbSP_FertilityLow			:_Domoticz_SwitchPoint;
	fbEI_FertilityLow			:Domoticz_ErrorInterface;
END_VAR

IF __ISVALIDREF(scConnector) THEN
	Main();
END_IF

ACTION Main:
{attribute 'conditionalshow'}
//Call parent function
SUPER^.Main();

//Call all functions
//Data timeout update rate is set by user, default 60m
afb_ObjectReal_Out[1].tDataTimeOut := TO_TIME(TO_UDINT(tUpdateRate)*2);
afb_ObjectReal_Out[1](scConnector := scConnector, 		uiIdentifier := uiIdentifier_Temperature, 		rxUpdateInterlock := rxUpdateInterlock_int,			rValueAct => rTemperature);

afb_ObjectReal_Out[2].tDataTimeOut := TO_TIME(TO_UDINT(tUpdateRate)*2);
afb_ObjectReal_Out[2](scConnector := scConnector, 		uiIdentifier := uiIdentifier_Moisture, 			rxUpdateInterlock := rxUpdateInterlock_int,			rValueAct => rMoisture);

afb_ObjectReal_Out[3].tDataTimeOut := TO_TIME(TO_UDINT(tUpdateRate)*2);
afb_ObjectReal_Out[3](scConnector := scConnector, 		uiIdentifier := uiIdentifier_Light, 			rxUpdateInterlock := rxUpdateInterlock_int,			rValueAct => rLux);

afb_ObjectReal_Out[4].tDataTimeOut := TO_TIME(TO_UDINT(tUpdateRate)*2);
afb_ObjectReal_Out[4](scConnector := scConnector, 		uiIdentifier := uiIdentifier_Fertility, 		rxUpdateInterlock := rxUpdateInterlock_int,			rValueAct => rFertility);

afb_ObjectBool_InOut[1].eCommandType := _Domoticz_eCommandType.SwitchLight;
afb_ObjectBool_InOut[1](scConnector := scConnector,		uiIdentifier := uiIdentifier_UpdateSwitch,		rxUpdateInterlock := rxUpdateInterlock_int,			xValueSet := xTONUpdate);

//Give plugin time to read data (limit time), only if specified
IF tUpdateRate < T#5M 
AND uiIdentifier_UpdateSwitch <> 0 THEN 
	tUpdateRate := T#5M; 
END_IF

//Timer
TON_Update(IN := NOT TON_Update.Q, PT := tUpdateRate);
IF TON_Update.Q THEN
	xTONUpdate := NOT xTONUpdate;
END_IF

//Errors
//********************************************DATA
fbEI_DataTimeOut.sInstanceName := sInstanceName;
fbEI_DataTimeOut.tErrorDelay := T#500MS;	//Give objects TIME TO be overruled BY other updates
fbEI_DataTimeOut(
	scConnector:= scConnector,
	xError:= xDataTimeOut_int
			AND (afb_ObjectReal_Out[1].xDataTimedOut
			OR afb_ObjectReal_Out[2].xDataTimedOut
			OR afb_ObjectReal_Out[3].xDataTimedOut
			OR afb_ObjectReal_Out[4].xDataTimedOut),
	eErrorID:= Domoticz_eErrors.ObjectDataTimeOut
);

//********************************************MOISTURE
fbSP_MoistureLow(
	xEnable:= rMoisture > 0,
	rInput:= rMoisture, 
	rSwitchPoint:= rThresholdMoistureLow_int, 
	rHysteresis:= 100, 
	xInvert:= TRUE, 
	xOut=> );
fbEI_MoistureLow.sInstanceName := sInstanceName;
fbEI_MoistureLow.sErrorInfo := TO_STRING(TO_INT(_Domoticz_RoundDecimals(rMoisture,0)));
fbEI_MoistureLow.sErrorInfo := CONCAT(fbEI_MoistureLow.sErrorInfo, ' %');
fbEI_MoistureLow(
	scConnector:= scConnector,
	xError:= fbSP_MoistureLow.xOut 
			AND rThresholdMoistureLow_int > 0
			AND uiIdentifier_Moisture > 0,
	eErrorID:= Domoticz_eErrors.MiFlora_MoistureLow
);

//********************************************FERTILITY
fbSP_FertilityLow(
	xEnable:= rFertility > 0,
	rInput:= rFertility, 
	rSwitchPoint:= rThresholdFertilityLow_int, 
	rHysteresis:= 100, 
	xInvert:= TRUE, 
	xOut=> );
fbEI_FertilityLow.sInstanceName := sInstanceName;
fbEI_FertilityLow.sErrorInfo := TO_STRING(TO_INT(_Domoticz_RoundDecimals(rFertility,0)));
fbEI_FertilityLow.sErrorInfo := CONCAT(fbEI_FertilityLow.sErrorInfo, ' uS/cm');
fbEI_FertilityLow(
	scConnector:= scConnector,
	xError:= fbSP_FertilityLow.xOut 
			AND rThresholdFertilityLow_int > 0 
			AND uiIdentifier_Fertility > 0,
	eErrorID:= Domoticz_eErrors.MiFlora_FertilityLow
);
END_ACTION

{attribute 'monitoring' := 'call'} PROPERTY rThresholdMoistureLow :REAL
SET
rThresholdMoistureLow_int := rThresholdMoistureLow;
END_SET
GET
rThresholdMoistureLow := rThresholdMoistureLow_int;
END_GET
END_PROPERTY

{attribute 'monitoring' := 'call'} PROPERTY rThresholdFertilityLow :REAL
SET
rThresholdFertilityLow_int := rThresholdFertilityLow;
END_SET
GET
rThresholdFertilityLow := rThresholdFertilityLow_int;
END_GET
END_PROPERTY

END_FUNCTION_BLOCK

// Function Blocks/Server/Domoticz_Server
{attribute 'conditionalshow_all_locals'}
FUNCTION_BLOCK Domoticz_Server EXTENDS _Domoticz_Server
VAR_OUTPUT
END_VAR
VAR
END_VAR

{attribute 'conditionalshow'}
//Call parent function
SUPER^.Main();

END_FUNCTION_BLOCK

// Function Blocks/Hardware/System/Network/Domoticz_SpeedTest
{attribute 'conditionalshow_all_locals'}
FUNCTION_BLOCK Domoticz_SpeedTest EXTENDS _Domoticz_Connector_Out
VAR_INPUT
	uiIdentifier_Ping			:UINT;	//Ping time
	uiIdentifier_Download		:UINT;	//Download speed
	uiIdentifier_Upload			:UINT;	//Upload speed
	tUpdateRate					:TIME := T#60M;	//Used for data timeout
END_VAR
VAR_OUTPUT
	tPing						:TIME;
	rDownload					:REAL;
	rUpload						:REAL;
END_VAR
VAR
	afb_ObjectReal_Out			:ARRAY[1..3] OF _Domoticz_ObjectReal_Out;
	
	tThresholdPingHigh_int		:TIME := T#30MS;	//ms
	fbSP_PingHigh				:_Domoticz_SwitchPoint;
	fbEI_PingHigh				:Domoticz_ErrorInterface;
	
	rThresholdDownloadSpeedLow_int	:REAL := 100;
	fbSP_DownloadSpeedLow		:_Domoticz_SwitchPoint;
	fbEI_DownloadSpeedLow		:Domoticz_ErrorInterface;
	
	rThresholdUploadSpeedLow_int	:REAL := 10;
	fbSP_UploadSpeedLow			:_Domoticz_SwitchPoint;
	fbEI_UploadSpeedLow			:Domoticz_ErrorInterface;
END_VAR

IF __ISVALIDREF(scConnector) THEN
	Main();
END_IF

ACTION Main:
{attribute 'conditionalshow'}
//Call parent function
SUPER^.Main();

//Call all functions
//Data timeout (update rate is set by user, default 60m)
afb_ObjectReal_Out[1].tDataTimeOut := TO_TIME(TO_UDINT(tUpdateRate)*4);
afb_ObjectReal_Out[1](scConnector := scConnector, 	uiIdentifier := uiIdentifier_Ping,		rxUpdateInterlock := rxUpdateInterlock_int);

afb_ObjectReal_Out[2].tDataTimeOut := TO_TIME(TO_UDINT(tUpdateRate)*4);
afb_ObjectReal_Out[2](scConnector := scConnector, 	uiIdentifier := uiIdentifier_Download, 	rxUpdateInterlock := rxUpdateInterlock_int,			rValueAct => rDownload);

afb_ObjectReal_Out[3].tDataTimeOut := TO_TIME(TO_UDINT(tUpdateRate)*4);
afb_ObjectReal_Out[3](scConnector := scConnector, 	uiIdentifier := uiIdentifier_Upload, 	rxUpdateInterlock := rxUpdateInterlock_int,			rValueAct => rUpload);
tPing := TO_TIME(afb_ObjectReal_Out[1].rValueAct);								  
									  
//Errors
//********************************************DATA
fbEI_DataTimeOut.sInstanceName := sInstanceName;
fbEI_DataTimeOut.tErrorDelay := T#500MS;	//Give objects TIME TO be overruled BY other updates
fbEI_DataTimeOut(
	scConnector:= scConnector,
	xError:= xDataTimeOut_int
			AND (afb_ObjectReal_Out[1].xDataTimedOut
			OR afb_ObjectReal_Out[2].xDataTimedOut
			OR afb_ObjectReal_Out[3].xDataTimedOut),
	eErrorID:= Domoticz_eErrors.ObjectDataTimeOut
);

//********************************************PING
fbSP_PingHigh(
	xEnable:= tPing > T#0MS,
	rInput:= TO_REAL(tPing), 
	rSwitchPoint:= TO_REAL(tThresholdPingHigh_int), 
	rHysteresis:= 10, 
	xInvert:= FALSE, 
	xOut=> );
fbEI_PingHigh.sInstanceName := sInstanceName;
fbEI_PingHigh.sErrorInfo := TO_STRING(tPing);
fbEI_PingHigh.sErrorInfo := CONCAT(fbEI_PingHigh.sErrorInfo, ' ms');
fbEI_PingHigh(
	scConnector:= scConnector,
	xError:= fbSP_PingHigh.xOut
			AND tThresholdPingHigh_int > T#0MS
			AND uiIdentifier_Ping > 0,
	eErrorID:= Domoticz_eErrors.SpeedTest_PingHigh
);

//********************************************DOWNLOAD
fbSP_DownloadSpeedLow(
	xEnable:= rDownload > 0,
	rInput:= rDownload, 
	rSwitchPoint:= rThresholdDownloadSpeedLow_int, 
	rHysteresis:= 10, 
	xInvert:= TRUE, 
	xOut=> );
fbEI_DownloadSpeedLow.sInstanceName := sInstanceName;
fbEI_DownloadSpeedLow.sErrorInfo := TO_STRING(_Domoticz_RoundDecimals(rDownload,1));
fbEI_DownloadSpeedLow.sErrorInfo := CONCAT(fbEI_DownloadSpeedLow.sErrorInfo, ' Mb/s');
fbEI_DownloadSpeedLow(
	scConnector:= scConnector,
	xError:= fbSP_DownloadSpeedLow.xOut 
			AND rThresholdDownloadSpeedLow_int > 0
			AND uiIdentifier_Download > 0,
	eErrorID:= Domoticz_eErrors.SpeedTest_DownloadSpeedLow
);

//********************************************UPLOAD
fbSP_UploadSpeedLow(
	xEnable:= rUpload > 0,
	rInput:= rUpload, 
	rSwitchPoint:= rThresholdUploadSpeedLow_int, 
	rHysteresis:= 10, 
	xInvert:= TRUE, 
	xOut=> );
fbEI_UploadSpeedLow.sInstanceName := sInstanceName;
fbEI_UploadSpeedLow.sErrorInfo := TO_STRING(_Domoticz_RoundDecimals(rUpload,1));
fbEI_UploadSpeedLow.sErrorInfo := CONCAT(fbEI_UploadSpeedLow.sErrorInfo, ' Mb/s');
fbEI_UploadSpeedLow(
	scConnector:= scConnector,
	xError:= fbSP_UploadSpeedLow.xOut 
			AND rThresholdUploadSpeedLow_int > 0 
			AND uiIdentifier_Upload > 0,
	eErrorID:= Domoticz_eErrors.SpeedTest_UploadSpeedLow
);
END_ACTION

{attribute 'monitoring' := 'call'} PROPERTY tThresholdPingHigh :TIME
SET
tThresholdPingHigh_int := tThresholdPingHigh;
END_SET
GET
tThresholdPingHigh := tThresholdPingHigh_int;
END_GET
END_PROPERTY

{attribute 'monitoring' := 'call'} PROPERTY rThresholdDownloadSpeedLow :REAL
SET
rThresholdDownloadSpeedLow_int := rThresholdDownloadSpeedLow;
END_SET
GET
rThresholdDownloadSpeedLow := rThresholdDownloadSpeedLow_int;
END_GET
END_PROPERTY

{attribute 'monitoring' := 'call'} PROPERTY rThresholdUploadSpeedLow :REAL
SET
rThresholdUploadSpeedLow_int := rThresholdUploadSpeedLow;
END_SET
GET
rThresholdUploadSpeedLow := rThresholdUploadSpeedLow_int;
END_GET
END_PROPERTY

END_FUNCTION_BLOCK

// Function Blocks/Hardware/Custom/Domoticz_CustomDimmer
{attribute 'conditionalshow_all_locals'}
FUNCTION_BLOCK Domoticz_CustomDimmer EXTENDS _Domoticz_Connector_InOut_Extended
VAR_INPUT
	uiIdentifier				:UINT;	//Device to control
	xEnable						:BOOL;
	byValue_Set					:BYTE;
END_VAR
VAR_OUTPUT
	xEnabled					:BOOL;
	byValue_Act					:BYTE;
END_VAR
VAR
	afb_ObjectBool_InOut		:ARRAY[1..1] OF _Domoticz_ObjectBool_InOut;
	afb_ObjectInt_InOut			:ARRAY[1..1] OF _Domoticz_ObjectInt_InOut;
	xUseOnlyNValue_int			:BOOL := FALSE;
END_VAR

IF __ISVALIDREF(scConnector) THEN
	Main();
END_IF

ACTION Main:
{attribute 'conditionalshow'}
//Call parent function
SUPER^.Main();

//Call all functions
afb_ObjectBool_InOut[1].tDataTimeOut := tDataTimeOut_int;
afb_ObjectBool_InOut[1](scConnector := scConnector, 	uiIdentifier := uiIdentifier, 	rxUpdateInterlock := rxUpdateInterlock_int,	 	xValueSet := xEnable, 		xValueAct => xEnabled);

afb_ObjectInt_InOut[1].tDataTimeOut := tDataTimeOut_int;
afb_ObjectInt_InOut[1].xUseOnlyNValue := xUseOnlyNValue_int;
afb_ObjectInt_InOut[1](	scConnector := scConnector, 	uiIdentifier := uiIdentifier,	rxUpdateInterlock := rxUpdateInterlock_int,	 	iValueSet := byValue_Set);

//Set value to zero if not enabled, else pass-through
IF NOT xEnabled AND NOT xUseOnlyNValue THEN 
	byValue_Act := TO_BYTE(afb_ObjectInt_InOut[1].iValueSetLimitLow); 
ELSE
	byValue_Act := TO_BYTE(afb_ObjectInt_InOut[1].iValueAct);
END_IF

//Force status if enabled
IF xForceSetValues AND xEnable <> xEnabled AND NOT xUseOnlyNValue THEN
	afb_ObjectBool_InOut[1].ForceSet(tForceSetValues_int);
ELSIF xForceSetValues AND (xEnabled OR xUseOnlyNValue) AND byValue_Set <> byValue_Act THEN
	afb_ObjectInt_InOut[1].ForceSet(tForceSetValues_int);
END_IF

//Errors
fbEI_DataTimeOut.sInstanceName := sInstanceName;
fbEI_DataTimeOut.tErrorDelay := T#500MS;	//Give objects TIME TO be overruled BY other updates
fbEI_DataTimeOut(
	scConnector:= scConnector,
	xError:= xDataTimeOut_int
			AND (afb_ObjectBool_InOut[1].xDataTimedOut
			OR afb_ObjectInt_InOut[1].xDataTimedOut),
	eErrorID:= Domoticz_eErrors.ObjectDataTimeOut
);
END_ACTION

{attribute 'monitoring' := 'call'} PROPERTY xUseOnlyNValue :BOOL
SET
xUseOnlyNValue_int := xUseOnlyNValue;
END_SET
GET
xUseOnlyNValue := xUseOnlyNValue_int;
END_GET
END_PROPERTY

END_FUNCTION_BLOCK

// Function Blocks/Hardware/Custom/Domoticz_CustomSwitch
{attribute 'conditionalshow_all_locals'}
FUNCTION_BLOCK Domoticz_CustomSwitch EXTENDS _Domoticz_Connector_InOut_Extended
VAR_INPUT
	uiIdentifier				:UINT;	//Device to control
	xEnable						:BOOL;
END_VAR
VAR_OUTPUT
	xEnabled					:BOOL;
END_VAR
VAR
	afb_ObjectBool_InOut		:ARRAY[1..1] OF _Domoticz_ObjectBool_InOut;
	xInvert_int					:BOOL;	//Invert xEnable/xEnabled
END_VAR

IF __ISVALIDREF(scConnector) THEN
	Main();
END_IF

ACTION Main:
{attribute 'conditionalshow'}
//Call parent function
SUPER^.Main();

//Call all functions
afb_ObjectBool_InOut[1].tDataTimeOut := tDataTimeOut_int;
afb_ObjectBool_InOut[1].eCommandType := _Domoticz_eCommandType.SwitchLight;
afb_ObjectBool_InOut[1](scConnector := scConnector, 	uiIdentifier := uiIdentifier, 	xValueSet := (xEnable XOR xInvert_int));

//Set output
xEnabled := afb_ObjectBool_InOut[1].xValueAct XOR xInvert_int;

//Force status if enabled
IF xForceSetValues AND (xEnable XOR xInvert_int) <> (xEnabled XOR xInvert_int) THEN
	afb_ObjectBool_InOut[1].ForceSet(tForceSetValues_int);
END_IF

//Errors
fbEI_DataTimeOut.sInstanceName := sInstanceName;
fbEI_DataTimeOut.tErrorDelay := T#500MS;	//Give objects TIME TO be overruled BY other updates
fbEI_DataTimeOut(
	scConnector:= scConnector,
	xError:= xDataTimeOut_int
			AND (afb_ObjectBool_InOut[1].xDataTimedOut),
	eErrorID:= Domoticz_eErrors.ObjectDataTimeOut
);
END_ACTION

{attribute 'monitoring' := 'call'} PROPERTY xInvert :BOOL
SET
xInvert_int := xInvert;
END_SET
GET
xInvert := xInvert_int;
END_GET
END_PROPERTY

END_FUNCTION_BLOCK

// Function Blocks/Hardware/Custom/Domoticz_CustomSensor
{attribute 'conditionalshow_all_locals'}
FUNCTION_BLOCK Domoticz_CustomSensor EXTENDS _Domoticz_Connector_InOut_Extended
VAR_INPUT
	uiIdentifier				:UINT;	//Device to control
	rValueSet					:REAL;
	
END_VAR
VAR_OUTPUT
	rValueAct					:REAL;
END_VAR
VAR
	afb_ObjectReal_InOut		:ARRAY[1..1] OF _Domoticz_ObjectReal_InOut;
	rSet,rAct					:REAL; //Calculate set/act value with scaling for forcing
	rScalingSet_int				:REAL := 1;
	rScalingAct_int				:REAL := 1;
END_VAR

IF __ISVALIDREF(scConnector) THEN
	Main();
END_IF

ACTION Main:
{attribute 'conditionalshow'}
//Call parent function
SUPER^.Main();

//Filter set value, filter on two decimals
rSet := _Domoticz_RoundDecimals((rValueSet*rScalingSet_int),2);	//Don't use scaling of object because of decimals

//Call all functions
afb_ObjectReal_InOut[1].tDataTimeOut := tDataTimeOut_int;
afb_ObjectReal_InOut[1](scConnector := scConnector, 	uiIdentifier := uiIdentifier,		rValueSet := rSet,		rValueAct => rAct);
		
//Filter act value, filter on two deciamls				
rValueAct := _Domoticz_RoundDecimals((rAct*rScalingAct_int),2);	//Don't use scaling of object because of decimals

//Force status if enabled
IF xForceSetValues AND rSet <> rAct THEN
	afb_ObjectReal_InOut[1].ForceSet(tForceSetValues_int);
END_IF

//Errors
fbEI_DataTimeOut.sInstanceName := sInstanceName;
fbEI_DataTimeOut.tErrorDelay := T#500MS;	//Give objects TIME TO be overruled BY other updates
fbEI_DataTimeOut(
	scConnector:= scConnector,
	xError:= xDataTimeOut_int
			AND (afb_ObjectReal_InOut[1].xDataTimedOut),
	eErrorID:= Domoticz_eErrors.ObjectDataTimeOut
);
END_ACTION

{attribute 'monitoring' := 'call'} PROPERTY rScalingSet :REAL
SET
rScalingSet_int := rScalingSet;
END_SET
GET
rScalingSet := rScalingSet_int;
END_GET
END_PROPERTY

{attribute 'monitoring' := 'call'} PROPERTY rScalingAct :REAL
SET
rScalingAct_int := rScalingAct;
END_SET
GET
rScalingAct := rScalingAct_int;
END_GET
END_PROPERTY

END_FUNCTION_BLOCK

// Function Blocks/Other/Domoticz_ServerLog
{attribute 'conditionalshow_all_locals'}
FUNCTION_BLOCK Domoticz_ServerLog EXTENDS _Domoticz_Connector
VAR_INPUT
	xEmptyLog			:BOOL;
	eFilter_Source		:_Domoticz_eDataSource;
	uiFilter_ID			:UINT;
END_VAR             	
VAR_OUTPUT          	
	ascObjectData		:ARRAY[1..Domoticz_Properties.uiInterfaceLog_MaxEntries] OF Domoticz_scObjectData;
END_VAR
VAR
	xNewObject_Rx_int	:BOOL;
	xNewObject_Tx_int	:BOOL;
	uiForLoop			:UINT;
	uiForLoop_Empty		:UINT;
END_VAR

IF __ISVALIDREF(scConnector) THEN
	Main();
END_IF

METHOD PRIVATE ShiftArray
VAR_INPUT
END_VAR
//Shift all data, throw away oldest one
FOR uiForLoop := (Domoticz_Properties.uiInterfaceLog_MaxEntries) TO 2 BY -1 DO
	ascObjectData[uiForLoop] := ascObjectData[uiForLoop-1];
END_FOR
END_METHOD

ACTION Main:
//Transmit data
IF scConnector.xNewObject_Tx AND NOT xNewObject_Tx_int
AND(eFilter_Source = _Domoticz_eDataSource.All OR eFilter_Source = _Domoticz_eDataSource.PLC)
AND (uiFilter_ID = scConnector.scObjectData_Tx.uiIdentifier OR uiFilter_ID = 0) THEN
	xNewObject_Tx_int := TRUE;
	ShiftArray();
	ascObjectData[1] := scConnector.scObjectData_Tx;
	ascObjectData[1].dtTimeStamp := scConnector.scTwilightData.dtSystem;	//Set timestamp, normally not given
	ascObjectData[1].eSource := _Domoticz_eDataSource.PLC;	//Overwrite source
ELSIF NOT scConnector.xNewObject_Tx AND xNewObject_Tx_int THEN
	xNewObject_Tx_int := FALSE;
	
//Receive data
ELSIF scConnector.xNewObject_Rx AND NOT xNewObject_Rx_int
AND (eFilter_Source = _Domoticz_eDataSource.All OR scConnector.scObjectData_Rx.eSource = eFilter_Source)
AND (uiFilter_ID = scConnector.scObjectData_Rx.uiIdentifier OR uiFilter_ID = 0) THEN
	xNewObject_Rx_int := TRUE;
	ShiftArray();
	ascObjectData[1] := scConnector.scObjectData_Rx;
ELSIF NOT scConnector.xNewObject_Rx AND xNewObject_Rx_int THEN
	xNewObject_Rx_int := FALSE;
END_IF

//Empty all entries
IF xEmptyLog THEN
	FOR uiForLoop := 1 TO Domoticz_Properties.uiInterfaceLog_MaxEntries DO
		ascObjectData[uiForLoop].uiIdentifier := 0;
		ascObjectData[uiForLoop].dtLastUpdate := DT#1970-1-1-0:0:0;
		ascObjectData[uiForLoop].dtTimeStamp := DT#1970-1-1-0:0:0;
		ascObjectData[uiForLoop].eSource := _Domoticz_eDataSource.All;
		ascObjectData[uiForLoop].eCommand := _Domoticz_eCommandType.Default;
		ascObjectData[uiForLoop].iValue :=0;
		FOR uiForLoop_Empty := 1 TO Domoticz_Constants.uiMaxSValues DO
			ascObjectData[uiForLoop].asValue[uiForLoop_Empty] := '';
		END_FOR
		ascObjectData[uiForLoop].sDeviceType := '';
	END_FOR
END_IF
END_ACTION

END_FUNCTION_BLOCK

// Function Blocks/Hardware/Devices/Domoticz_Tasmota
{attribute 'conditionalshow_all_locals'}
FUNCTION_BLOCK Domoticz_Tasmota EXTENDS _Domoticz_Connector_InOut
VAR_INPUT
	uiIdentifier_Relay					:UINT;			//Relay control
	uiIdentifier_TempHumBaro			:UINT;			//Temperature / Humidity / Barometer
	uiIdentifier_Power					:UINT;			//Usage
	uiIdentifier_Illuminance			:UINT;			//Lux
	uiIdentifier_1um					:UINT;			//Particles 1 µm
	uiIdentifier_2_5um					:UINT;			//Particles 2.5 µm
	uiIdentifier_10um					:UINT;			//Particles 10 µm
	uiIdentifier_Voltage				:UINT;			//Voltage measured
	uiIdentifier_Current				:UINT;			//Current measured
	uiIdentifier_CarbonDioxide			:UINT;			//CO/CO2 (ppm)
	tUpdateRate							:TIME := T#60M;	//Used for data timeout
	xEnable								:BOOL;			//Relay
END_VAR                         		
VAR_OUTPUT                      		
	xEnabled							:BOOL;
	rTemperature						:REAL;
	rHumidity							:REAL;
	rBarometer							:REAL;
	rPowerUsageActual					:REAL;
	rPowerUsageToday					:REAL;
	rPowerUsageCumulative				:REAL;
	rIlluminance						:REAL;
	rParticles_1um						:REAL;
	rParticles_2_5um					:REAL;
	rParticles_10um						:REAL;
	rVoltage							:REAL;
	rCurrent							:REAL;
	rCarbonDioxide						:REAL;
END_VAR                         		
VAR	                            		
	afb_ObjectBool_InOut				:ARRAY[1..1] OF _Domoticz_ObjectBool_InOut;
	afb_ObjectReal_Out					:ARRAY[1..7] OF _Domoticz_ObjectReal_Out;
	afb_ObjectArrayReal_Out				:ARRAY[1..2] OF _Domoticz_ObjectArrayReal_Out;
	             
	rThresholdVoltage_int				:REAL := 200;        	
	fbEI_PowerFailure					:Domoticz_ErrorInterface;
	fbTON_PowerFailure_Enabled			:TON;
	
	//Temperature
	rThresholdTemperatureHigh_int		:REAL := 30;	//C
	fbSP_TemperatureHigh				:_Domoticz_SwitchPoint;
	fbEI_TemperatureHigh				:Domoticz_ErrorInterface;
	
	rThresholdTemperatureLow_int		:REAL := 15;	//C
	fbSP_TemperatureLow					:_Domoticz_SwitchPoint;
	fbEI_TemperatureLow					:Domoticz_ErrorInterface;
	
	//Humidity
	rThresholdHumidityHigh_int			:REAL := 70;	//%
	fbSP_HumidityHigh					:_Domoticz_SwitchPoint;
	fbEI_HumidityHigh					:Domoticz_ErrorInterface;
	
	rThresholdHumidityLow_int			:REAL := 30;	//%
	fbSP_HumidityLow					:_Domoticz_SwitchPoint;
	fbEI_HumidityLow					:Domoticz_ErrorInterface;
	
	//Power
	rThresholdPowerUsageToday_int		:REAL := 15.0; //kWh
	fbEI_PowerUsageToday				:Domoticz_ErrorInterface;
	
	rThresholdPowerUsageHigh_int		:REAL := 3000;
	fbSP_PowerUsageHigh					:_Domoticz_SwitchPoint;
	fbEI_PowerUsageHigh					:Domoticz_ErrorInterface;
	
	//Current
	rThresholdCurrentHigh_int			:REAL := 10;	//A
	fbSP_CurrentHigh					:_Domoticz_SwitchPoint;
	fbEI_CurrentHigh					:Domoticz_ErrorInterface;
	                            		
	rThresholdCurrentMax_int			:REAL := 14;	//A
	fbSP_CurrentMax						:_Domoticz_SwitchPoint;
	fbEI_CurrentMax						:Domoticz_ErrorInterface;
	
	//PM xx
	rThresholdParticlesHigh_1um_int		:REAL := 5;		//ug/m3
	fbSP_1umHigh						:_Domoticz_SwitchPoint;
	fbEI_1umHigh						:Domoticz_ErrorInterface;
	
	rThresholdParticlesHigh_2_5um_int	:REAL := 10;	//ug/m3
	fbSP_2_5umHigh						:_Domoticz_SwitchPoint;
	fbEI_2_5umHigh						:Domoticz_ErrorInterface;
	
	rThresholdParticlesHigh_10um_int	:REAL := 20;	//ug/m3
	fbSP_10umHigh						:_Domoticz_SwitchPoint;
	fbEI_10umHigh						:Domoticz_ErrorInterface;

	//Air Quality
	rThresholdCarbonDioxideHigh_int		:REAL := 2500;	//ppm
	fbSP_CarbonDioxideHigh				:_Domoticz_SwitchPoint;
	fbEI_CarbonDioxideHigh				:Domoticz_ErrorInterface;
	
	rThresholdCarbonDioxideCritical_int	:REAL := 5000;	//ppm
	fbSP_CarbonDioxideCritical			:_Domoticz_SwitchPoint;
	fbEI_CarbonDioxideCritical			:Domoticz_ErrorInterface;
END_VAR

IF __ISVALIDREF(scConnector) THEN
	Main();
END_IF

ACTION Main:
{attribute 'conditionalshow'}
//Call parent function
SUPER^.Main();

//Call all functions
//Data timeout update rate is set by user, default 60m
afb_ObjectBool_InOut[1].tDataTimeOut := TO_TIME(TO_UDINT(tUpdateRate)*2);
afb_ObjectBool_InOut[1].eCommandType := _Domoticz_eCommandType.SwitchLight;
afb_ObjectBool_InOut[1](scConnector := scConnector, 	uiIdentifier := uiIdentifier_Relay, 		rxUpdateInterlock := rxUpdateInterlock_int,			xValueSet := xEnable, 	xValueAct => xEnabled);

afb_ObjectReal_Out[1].tDataTimeOut := TO_TIME(TO_UDINT(tUpdateRate)*2);
afb_ObjectReal_Out[1](	scConnector := scConnector, 	uiIdentifier := uiIdentifier_Illuminance, 	rxUpdateInterlock := rxUpdateInterlock_int,			rValueAct => rIlluminance);

afb_ObjectReal_Out[2].tDataTimeOut := TO_TIME(TO_UDINT(tUpdateRate)*2);
afb_ObjectReal_Out[2].eDataSource := _Domoticz_eDataSource.HTTP;     
afb_ObjectReal_Out[2](	scConnector := scConnector, 	uiIdentifier := uiIdentifier_1um, 			rxUpdateInterlock := rxUpdateInterlock_int,			rValueAct => rParticles_1um);
                                                                                                	
afb_ObjectReal_Out[3].tDataTimeOut := TO_TIME(TO_UDINT(tUpdateRate)*2);   
afb_ObjectReal_Out[3].eDataSource := _Domoticz_eDataSource.HTTP;                           	
afb_ObjectReal_Out[3](	scConnector := scConnector, 	uiIdentifier := uiIdentifier_2_5um, 		rxUpdateInterlock := rxUpdateInterlock_int,			rValueAct => rParticles_2_5um);
                                                                                                	
afb_ObjectReal_Out[4].tDataTimeOut := TO_TIME(TO_UDINT(tUpdateRate)*2);  
afb_ObjectReal_Out[4].eDataSource := _Domoticz_eDataSource.HTTP;                       	
afb_ObjectReal_Out[4](	scConnector := scConnector, 	uiIdentifier := uiIdentifier_10um, 			rxUpdateInterlock := rxUpdateInterlock_int,			rValueAct => rParticles_10um);
                                                                                                	
afb_ObjectReal_Out[5].tDataTimeOut := TO_TIME(TO_UDINT(tUpdateRate)*2);                         	
afb_ObjectReal_Out[5](	scConnector := scConnector, 	uiIdentifier := uiIdentifier_Voltage, 		rxUpdateInterlock := rxUpdateInterlock_int,			rValueAct => rVoltage);
                                                                                                	
afb_ObjectReal_Out[6].tDataTimeOut := TO_TIME(TO_UDINT(tUpdateRate)*2);                         	
afb_ObjectReal_Out[6](	scConnector := scConnector, 	uiIdentifier := uiIdentifier_Current, 		rxUpdateInterlock := rxUpdateInterlock_int,			rValueAct => rCurrent);
                                                                                                	
afb_ObjectReal_Out[7].tDataTimeOut := TO_TIME(TO_UDINT(tUpdateRate)*2);                         	
afb_ObjectReal_Out[7](	scConnector := scConnector, 	uiIdentifier := uiIdentifier_CarbonDioxide,	rxUpdateInterlock := rxUpdateInterlock_int,			rValueAct => rCarbonDioxide);

afb_ObjectArrayReal_Out[1].tDataTimeOut := TO_TIME(TO_UDINT(tUpdateRate)*2);
afb_ObjectArrayReal_Out[1](scConnector := scConnector, 	uiIdentifier := uiIdentifier_TempHumBaro,	rxUpdateInterlock := rxUpdateInterlock_int);

afb_ObjectArrayReal_Out[2].tDataTimeOut := TO_TIME(TO_UDINT(tUpdateRate)*2);
afb_ObjectArrayReal_Out[2](scConnector := scConnector, 	uiIdentifier := uiIdentifier_Power,			rxUpdateInterlock := rxUpdateInterlock_int);

//Output arrays
rTemperature			:= afb_ObjectArrayReal_Out[1].arValueAct[Domoticz_eSValues_TempHumBaro.Temperature];
rHumidity				:= afb_ObjectArrayReal_Out[1].arValueAct[Domoticz_eSValues_TempHumBaro.Humidity];
rBarometer				:= afb_ObjectArrayReal_Out[1].arValueAct[Domoticz_eSValues_TempHumBaro.Barometer];

rPowerUsageActual 		:= afb_ObjectArrayReal_Out[2].arValueAct[Domoticz_eSValues_Usage.Usage];
rPowerUsageCumulative	:= afb_ObjectArrayReal_Out[2].arValueAct[Domoticz_eSValues_Usage.UsageCumulative];
rPowerUsageToday		:= afb_ObjectArrayReal_Out[2].arValueAct[Domoticz_eSValues_Usage.UsageToday];

//Force status if enabled
IF xForceSetValues AND xEnable <> xEnabled THEN
	afb_ObjectBool_InOut[1].ForceSet(tForceSetValues_int);
END_IF

//Errors
//********************************************DATA
fbEI_DataTimeOut.sInstanceName := sInstanceName;
fbEI_DataTimeOut.tErrorDelay := T#500MS;	//Give objects TIME TO be overruled BY other updates
fbEI_DataTimeOut(
	scConnector:= scConnector,
	xError:= xDataTimeOut_int
			AND (afb_ObjectBool_InOut[1].xDataTimedOut
			OR afb_ObjectReal_Out[1].xDataTimedOut
			OR afb_ObjectReal_Out[2].xDataTimedOut
			OR afb_ObjectReal_Out[3].xDataTimedOut
			OR afb_ObjectReal_Out[4].xDataTimedOut
			OR afb_ObjectReal_Out[5].xDataTimedOut
			OR afb_ObjectReal_Out[6].xDataTimedOut
			OR afb_ObjectArrayReal_Out[1].xDataTimedOut
			OR afb_ObjectArrayReal_Out[2].xDataTimedOut),
	eErrorID:= Domoticz_eErrors.ObjectDataTimeOut
);

//********************************************POWER FAILURE
fbEI_PowerFailure.sInstanceName := sInstanceName;
fbEI_PowerFailure.sErrorInfo := TO_STRING(TO_INT(_Domoticz_RoundDecimals(rVoltage,0)));
fbEI_PowerFailure.sErrorInfo := CONCAT(fbEI_PowerFailure.sErrorInfo, ' V / ');
fbEI_PowerFailure.sErrorInfo := CONCAT(fbEI_PowerFailure.sErrorInfo, TO_STRING(TO_INT(_Domoticz_RoundDecimals(rPowerUsageActual,0))));
fbEI_PowerFailure.sErrorInfo := CONCAT(fbEI_PowerFailure.sErrorInfo, ' W');
fbEI_PowerFailure(
	scConnector:= scConnector,
	xError:= (rVoltage < rThresholdVoltage_int) AND (uiIdentifier_Voltage > 0) 
			AND fbTON_PowerFailure_Enabled.Q,	//Actual current not taken into account because connected devices can be turned off and not use any power.
	eErrorID:= Domoticz_eErrors.Tasmota_PowerFailure
);
fbTON_PowerFailure_Enabled(IN:=xEnabled, PT:=T#10M);	//It can take a while before readings are send to Domoticz

//********************************************USAGE TODAY
fbEI_PowerUsageToday.sInstanceName := sInstanceName;
fbEI_PowerUsageToday.sErrorInfo := TO_STRING(_Domoticz_RoundDecimals(rPowerUsageToday,2));
fbEI_PowerUsageToday.sErrorInfo := CONCAT(fbEI_PowerUsageToday.sErrorInfo, ' kWh');
fbEI_PowerUsageToday(
	scConnector:= scConnector,
	xError:= (rPowerUsageToday > rThresholdPowerUsageToday_int) AND uiIdentifier_Power > 0,
	eErrorID:= Domoticz_eErrors.Tasmota_PowerUsageToday
);

//********************************************USAGE
fbSP_PowerUsageHigh(
	xEnable:= rPowerUsageActual > 0,
	rInput:= rPowerUsageActual, 
	rSwitchPoint:= rThresholdPowerUsageHigh_int, 
	rHysteresis:= 500, 
	xInvert:= FALSE, 
	xOut=> );
fbEI_PowerUsageHigh.sInstanceName := sInstanceName;
fbEI_PowerUsageHigh.sErrorInfo := TO_STRING(TO_INT(_Domoticz_RoundDecimals(rPowerUsageActual,0)));
fbEI_PowerUsageHigh.sErrorInfo := CONCAT(fbEI_PowerUsageHigh.sErrorInfo, ' W');
fbEI_PowerUsageHigh(
	scConnector:= scConnector,
	xError:= fbSP_PowerUsageHigh.xOut 
			AND rThresholdPowerUsageHigh_int > 0
			AND uiIdentifier_Power > 0,
	eErrorID:= Domoticz_eErrors.Tasmota_PowerUsageHigh
);

//********************************************CURRENT
fbSP_CurrentHigh(
	xEnable:= rCurrent > 0,
	rInput:= rCurrent, 
	rSwitchPoint:= rThresholdCurrentHigh_int, 
	rHysteresis:= 2, 
	xInvert:= FALSE, 
	xOut=> );
fbEI_CurrentHigh.sInstanceName := sInstanceName;
fbEI_CurrentHigh.sErrorInfo := TO_STRING(_Domoticz_RoundDecimals(rCurrent,1));
fbEI_CurrentHigh.sErrorInfo := CONCAT(fbEI_CurrentHigh.sErrorInfo, ' A');
fbEI_CurrentHigh(
	scConnector:= scConnector,
	xError:= fbSP_CurrentHigh.xOut 
			AND rThresholdCurrentHigh_int > 0
			AND uiIdentifier_Current > 0,
	eErrorID:= Domoticz_eErrors.Tasmota_CurrentHigh
);

fbSP_CurrentMax(
	xEnable:= rCurrent > 0,
	rInput:= rCurrent, 
	rSwitchPoint:= rThresholdCurrentMax_int, 
	rHysteresis:= 2, 
	xInvert:= FALSE, 
	xOut=> );
fbEI_CurrentMax.sInstanceName := sInstanceName;
fbEI_CurrentMax.sErrorInfo := TO_STRING(_Domoticz_RoundDecimals(rCurrent,1));
fbEI_CurrentMax.sErrorInfo := CONCAT(fbEI_CurrentMax.sErrorInfo, ' A');
fbEI_CurrentMax(
	scConnector:= scConnector,
	xError:= fbSP_CurrentMax.xOut 
			AND rThresholdCurrentMax_int > 0
			AND uiIdentifier_Current > 0,
	eErrorID:= Domoticz_eErrors.Tasmota_CurrentMax
);

//********************************************TEMPERATURE
fbSP_TemperatureHigh(
	xEnable:= TRUE,		//rTemperature > 0,			//Temperature can drop below 0C
	rInput:= rTemperature, 
	rSwitchPoint:= rThresholdTemperatureHigh_int, 
	rHysteresis:= 3, 
	xInvert:= FALSE, 
	xOut=> );
fbEI_TemperatureHigh.sInstanceName := sInstanceName;
fbEI_TemperatureHigh.sErrorInfo := TO_STRING(_Domoticz_RoundDecimals(rTemperature,1));
fbEI_TemperatureHigh.sErrorInfo := CONCAT(fbEI_TemperatureHigh.sErrorInfo, ' C');
fbEI_TemperatureHigh(
	scConnector:= scConnector,
	xError:= fbSP_TemperatureHigh.xOut 
			AND rThresholdTemperatureHigh_int > 0
			AND uiIdentifier_TempHumBaro > 0,
	eErrorID:= Domoticz_eErrors.Tasmota_TemperatureHigh
);

